Fanuc TP program (LS listing): hosenrohr_oVersatz.ls

/PROG  hosenrohr_oVersatz
/ATTR
COMMENT	= "19-03-19 17:34:17";
PROG_SIZE	= 0;
DEFAULT_GROUP	= 1, *, *, *, *;
/APPL
    ARC Welding Equipment: 1, *, *, *, *;
/MN
   1:  CALL HOME_ALL;
   1:  UFRAME_NUM = 1;
   1:  UTOOL_NUM = 3;
   1:  COL GUARD ADJUST 150;
   1:  PR[91] = PR[90];
   1:  PR[91,1] = PR[90,1] + 0.213;
   1:  PR[91,2] = PR[90,2] + 0.028;
   1:  PR[91,3] = PR[90,3] + 1.330;
   1:  PR[92] = PR[91];
   1:  PR[92,3] = PR[92,3] + 50;
   1:J PR[92] 10% FINE;
   1:L PR[91] R[100]mm/sec CNT100;
   1:  CALL LASER_DRAHT_START;
   1:  PR[91,1] = PR[90,1] + 0.684;
   1:  PR[91,2] = PR[90,2] + -0.011;
   1:L PR[91] R[100]mm/sec CNT100;
   1:  PR[91,1] = PR[90,1] + 1.247;
   1:  PR[91,2] = PR[90,2] + -0.156;
   1:  PR[91,3] = PR[90,3] + 0.003;
   1:L PR[91] R[100]mm/sec CNT100;
   1:  PR[91,1] = PR[90,1] + 1.774;
   1:  PR[91,2] = PR[90,2] + -0.407;
   1:  PR[91,3] = PR[90,3] + 0.006;
   1:L PR[91] R[100]mm/sec CNT100;
   1:  PR[91,1] = PR[90,1] + 2.182;
   1:  PR[91,2] = PR[90,2] + -0.695;
   1:  PR[91,3] = PR[90,3] + 0.010;
   1:L PR[91] R[100]mm/sec CNT100;
   1:  PR[91,1] = PR[90,1] + 2.537;
   1:  PR[91,2] = PR[90,2] + -1.047;
   1:  PR[91,3] = PR[90,3] + 0.013;
   1:L PR[91] R[100]mm/sec CNT100;
   1:  PR[91,1] = PR[90,1] + 2.876;
   1:  PR[91,2] = PR[90,2] + -1.521;
   1:  PR[91,3] = PR[90,3] + 0.016;
   1:L PR[91] R[100]mm/sec CNT100;
   1:  PR[91,1] = PR[90,1] + 3.117;
   1:  PR[91,2] = PR[90,2] + -2.049;
   1:  PR[91,3] = PR[90,3] + 0.020;
   1:L PR[91] R[100]mm/sec CNT100;
   1:  PR[91,1] = PR[90,1] + 3.228;
   1:  PR[91,2] = PR[90,2] + -2.464;
   1:  PR[91,3] = PR[90,3] + 0.023;
   1:L PR[91] R[100]mm/sec CNT100;
   1:  PR[91,1] = PR[90,1] + 3.332;
   1:  PR[91,2] = PR[90,2] + -2.996;
   1:  PR[91,3] = PR[90,3] + 0.026;
   1:L PR[91] R[100]mm/sec CNT100;
   1:  PR[91,1] = PR[90,1] + 3.499;
   1:  PR[91,2] = PR[90,2] + -3.723;
   1:  PR[91,3] = PR[90,3] + 0.029;
   1:L PR[91] R[100]mm/sec CNT100;
   1:  PR[91,1] = PR[90,1] + 3.811;
   1:  PR[91,2] = PR[90,2] + -4.797;
   1:  PR[91,3] = PR[90,3] + 0.034;
   1:L PR[91] R[100]mm/sec CNT100;
   1:  PR[91,1] = PR[90,1] + 4.268;
   1:  PR[91,2] = PR[90,2] + -6.041;
   1:  PR[91,3] = PR[90,3] + 0.040;
   1:L PR[91] R[100]mm/sec CNT100;
   1:  PR[91,1] = PR[90,1] + 4.777;
   1:  PR[91,2] = PR[90,2] + -7.153;
   1:  PR[91,3] = PR[90,3] + 0.048;
   1:L PR[91] R[100]mm/sec CNT100;
   1:  PR[91,1] = PR[90,1] + 5.314;
   1:  PR[91,2] = PR[90,2] + -8.138;
   1:  PR[91,3] = PR[90,3] + 0.056;
   1:L PR[91] R[100]mm/sec CNT100;
   1:  PR[91,1] = PR[90,1] + 5.705;
   1:  PR[91,2] = PR[90,2] + -8.772;
   1:  PR[91,3] = PR[90,3] + 0.063;
   1:L PR[91] R[100]mm/sec CNT100;
   1:  PR[91,1] = PR[90,1] + 6.024;
   1:  PR[91,2] = PR[90,2] + -9.246;
   1:  PR[91,3] = PR[90,3] + 0.067;
   1:L PR[91] R[100]mm/sec CNT100;
   1:  PR[91,1] = PR[90,1] + 6.762;
   1:  PR[91,2] = PR[90,2] + -10.226;
   1:  PR[91,3] = PR[90,3] + 0.071;
   1:L PR[91] R[100]mm/sec CNT100;
   1:  PR[91,1] = PR[90,1] + 7.570;
   1:  PR[91,2] = PR[90,2] + -11.150;
   1:  PR[91,3] = PR[90,3] + 0.078;
   1:L PR[91] R[100]mm/sec CNT100;
   1:  PR[91,1] = PR[90,1] + 8.074;
   1:  PR[91,2] = PR[90,2] + -11.664;
   1:  PR[91,3] = PR[90,3] + 0.086;
   1:L PR[91] R[100]mm/sec CNT100;
   1:  PR[91,1] = PR[90,1] + 8.430;
   1:  PR[91,2] = PR[90,2] + -12.001;
   1:  PR[91,3] = PR[90,3] + 0.090;
   1:L PR[91] R[100]mm/sec CNT100;
   1:  PR[91,1] = PR[90,1] + 9.365;
   1:  PR[91,2] = PR[90,2] + -12.801;
   1:  PR[91,3] = PR[90,3] + 0.093;
   1:L PR[91] R[100]mm/sec CNT100;
   1:  PR[91,1] = PR[90,1] + 10.262;
   1:  PR[91,2] = PR[90,2] + -13.466;
   1:  PR[91,3] = PR[90,3] + 0.100;
   1:L PR[91] R[100]mm/sec CNT100;
   1:  PR[91,1] = PR[90,1] + 11.385;
   1:  PR[91,2] = PR[90,2] + -14.181;
   1:  PR[91,3] = PR[90,3] + 0.107;
   1:L PR[91] R[100]mm/sec CNT100;
   1:  PR[91,1] = PR[90,1] + 12.079;
   1:  PR[91,2] = PR[90,2] + -14.564;
   1:  PR[91,3] = PR[90,3] + 0.115;
   1:L PR[91] R[100]mm/sec CNT100;
   1:  PR[91,1] = PR[90,1] + 12.452;
   1:  PR[91,2] = PR[90,2] + -14.752;
   1:  PR[91,3] = PR[90,3] + 0.120;
   1:L PR[91] R[100]mm/sec CNT100;
   1:  PR[91,1] = PR[90,1] + 13.575;
   1:  PR[91,2] = PR[90,2] + -15.252;
   1:  PR[91,3] = PR[90,3] + 0.123;
   1:L PR[91] R[100]mm/sec CNT100;
   1:  PR[91,1] = PR[90,1] + 14.627;
   1:  PR[91,2] = PR[90,2] + -15.633;
   1:  PR[91,3] = PR[90,3] + 0.130;
   1:L PR[91] R[100]mm/sec CNT100;
   1:  PR[91,1] = PR[90,1] + 15.902;
   1:  PR[91,2] = PR[90,2] + -15.997;
   1:  PR[91,3] = PR[90,3] + 0.137;
   1:L PR[91] R[100]mm/sec CNT100;
   1:  PR[91,1] = PR[90,1] + 17.100;
   1:  PR[91,2] = PR[90,2] + -16.242;
   1:  PR[91,3] = PR[90,3] + 0.145;
   1:L PR[91] R[100]mm/sec CNT100;
   1:  PR[91,1] = PR[90,1] + 18.207;
   1:  PR[91,2] = PR[90,2] + -16.387;
   1:  PR[91,3] = PR[90,3] + 0.152;
   1:L PR[91] R[100]mm/sec CNT100;
   1:  PR[91,1] = PR[90,1] + 19.533;
   1:  PR[91,2] = PR[90,2] + -16.468;
   1:  PR[91,3] = PR[90,3] + 0.159;
   1:L PR[91] R[100]mm/sec CNT100;
   1:  PR[91,1] = PR[90,1] + 20.752;
   1:  PR[91,2] = PR[90,2] + -16.449;
   1:  PR[91,3] = PR[90,3] + 0.167;
   1:L PR[91] R[100]mm/sec CNT100;
   1:  PR[91,1] = PR[90,1] + 21.868;
   1:  PR[91,2] = PR[90,2] + -16.353;
   1:  PR[91,3] = PR[90,3] + 0.175;
   1:L PR[91] R[100]mm/sec CNT100;
   1:  PR[91,1] = PR[90,1] + 23.177;
   1:  PR[91,2] = PR[90,2] + -16.147;
   1:  PR[91,3] = PR[90,3] + 0.181;
   1:L PR[91] R[100]mm/sec CNT100;
   1:  PR[91,1] = PR[90,1] + 24.367;
   1:  PR[91,2] = PR[90,2] + -15.866;
   1:  PR[91,3] = PR[90,3] + 0.189;
   1:L PR[91] R[100]mm/sec CNT100;
   1:  PR[91,1] = PR[90,1] + 25.433;
   1:  PR[91,2] = PR[90,2] + -15.532;
   1:  PR[91,3] = PR[90,3] + 0.197;
   1:L PR[91] R[100]mm/sec CNT100;
   1:  PR[91,1] = PR[90,1] + 26.669;
   1:  PR[91,2] = PR[90,2] + -15.048;
   1:  PR[91,3] = PR[90,3] + 0.204;
   1:L PR[91] R[100]mm/sec CNT100;
   1:  PR[91,1] = PR[90,1] + 27.769;
   1:  PR[91,2] = PR[90,2] + -14.518;
   1:  PR[91,3] = PR[90,3] + 0.212;
   1:L PR[91] R[100]mm/sec CNT100;
   1:  PR[91,1] = PR[90,1] + 28.829;
   1:  PR[91,2] = PR[90,2] + -13.909;
   1:  PR[91,3] = PR[90,3] + 0.219;
   1:L PR[91] R[100]mm/sec CNT100;
   1:  PR[91,1] = PR[90,1] + 29.757;
   1:  PR[91,2] = PR[90,2] + -13.284;
   1:  PR[91,3] = PR[90,3] + 0.227;
   1:L PR[91] R[100]mm/sec CNT100;
   1:  PR[91,1] = PR[90,1] + 30.802;
   1:  PR[91,2] = PR[90,2] + -12.468;
   1:  PR[91,3] = PR[90,3] + 0.233;
   1:L PR[91] R[100]mm/sec CNT100;
   1:  PR[91,1] = PR[90,1] + 31.706;
   1:  PR[91,2] = PR[90,2] + -11.646;
   1:  PR[91,3] = PR[90,3] + 0.241;
   1:L PR[91] R[100]mm/sec CNT100;
   1:  PR[91,1] = PR[90,1] + 32.547;
   1:  PR[91,2] = PR[90,2] + -10.760;
   1:  PR[91,3] = PR[90,3] + 0.249;
   1:L PR[91] R[100]mm/sec CNT100;
   1:  PR[91,1] = PR[90,1] + 33.259;
   1:  PR[91,2] = PR[90,2] + -9.896;
   1:  PR[91,3] = PR[90,3] + 0.256;
   1:L PR[91] R[100]mm/sec CNT100;
   1:  PR[91,1] = PR[90,1] + 34.054;
   1:  PR[91,2] = PR[90,2] + -8.776;
   1:  PR[91,3] = PR[90,3] + 0.263;
   1:L PR[91] R[100]mm/sec CNT100;
   1:  PR[91,1] = PR[90,1] + 34.659;
   1:  PR[91,2] = PR[90,2] + -7.769;
   1:  PR[91,3] = PR[90,3] + 0.271;
   1:L PR[91] R[100]mm/sec CNT100;
   1:  PR[91,1] = PR[90,1] + 35.214;
   1:  PR[91,2] = PR[90,2] + -6.678;
   1:  PR[91,3] = PR[90,3] + 0.279;
   1:L PR[91] R[100]mm/sec CNT100;
   1:  PR[91,1] = PR[90,1] + 35.547;
   1:  PR[91,2] = PR[90,2] + -5.910;
   1:  PR[91,3] = PR[90,3] + 0.286;
   1:L PR[91] R[100]mm/sec CNT100;
   1:  PR[91,1] = PR[90,1] + 35.684;
   1:  PR[91,2] = PR[90,2] + -5.559;
   1:  PR[91,3] = PR[90,3] + 0.291;
   1:L PR[91] R[100]mm/sec CNT100;
   1:  PR[91,1] = PR[90,1] + 36.077;
   1:  PR[91,2] = PR[90,2] + -4.396;
   1:  PR[91,3] = PR[90,3] + 0.293;
   1:L PR[91] R[100]mm/sec CNT100;
   1:  PR[91,1] = PR[90,1] + 36.362;
   1:  PR[91,2] = PR[90,2] + -3.304;
   1:  PR[91,3] = PR[90,3] + 0.301;
   1:L PR[91] R[100]mm/sec CNT100;
   1:  PR[91,1] = PR[90,1] + 36.446;
   1:  PR[91,2] = PR[90,2] + -2.914;
   1:  PR[91,3] = PR[90,3] + 0.308;
   1:L PR[91] R[100]mm/sec CNT100;
   1:  PR[91,1] = PR[90,1] + 36.603;
   1:  PR[91,2] = PR[90,2] + -2.012;
   1:  PR[91,3] = PR[90,3] + 0.310;
   1:L PR[91] R[100]mm/sec CNT100;
   1:  PR[91,1] = PR[90,1] + 36.727;
   1:  PR[91,2] = PR[90,2] + -0.896;
   1:  PR[91,3] = PR[90,3] + 0.316;
   1:L PR[91] R[100]mm/sec CNT100;
   1:  PR[91,1] = PR[90,1] + 36.773;
   1:  PR[91,2] = PR[90,2] + -0.086;
   1:  PR[91,3] = PR[90,3] + 0.322;
   1:L PR[91] R[100]mm/sec CNT100;
   1:  PR[91,1] = PR[90,1] + 36.781;
   1:  PR[91,2] = PR[90,2] + 0.420;
   1:  PR[91,3] = PR[90,3] + 0.327;
   1:L PR[91] R[100]mm/sec CNT100;
   1:  PR[91,1] = PR[90,1] + 36.726;
   1:  PR[91,2] = PR[90,2] + 1.756;
   1:  PR[91,3] = PR[90,3] + 0.330;
   1:L PR[91] R[100]mm/sec CNT100;
   1:  PR[91,1] = PR[90,1] + 36.604;
   1:  PR[91,2] = PR[90,2] + 2.865;
   1:  PR[91,3] = PR[90,3] + 0.339;
   1:L PR[91] R[100]mm/sec CNT100;
   1:  PR[91,1] = PR[90,1] + 36.404;
   1:  PR[91,2] = PR[90,2] + 3.965;
   1:  PR[91,3] = PR[90,3] + 0.345;
   1:L PR[91] R[100]mm/sec CNT100;
   1:  PR[91,1] = PR[90,1] + 36.075;
   1:  PR[91,2] = PR[90,2] + 5.258;
   1:  PR[91,3] = PR[90,3] + 0.352;
   1:L PR[91] R[100]mm/sec CNT100;
   1:  PR[91,1] = PR[90,1] + 35.922;
   1:  PR[91,2] = PR[90,2] + 5.747;
   1:  PR[91,3] = PR[90,3] + 0.360;
   1:L PR[91] R[100]mm/sec CNT100;
   1:  PR[91,1] = PR[90,1] + 35.650;
   1:  PR[91,2] = PR[90,2] + 6.499;
   1:  PR[91,3] = PR[90,3] + 0.363;
   1:L PR[91] R[100]mm/sec CNT100;
   1:  PR[91,1] = PR[90,1] + 35.212;
   1:  PR[91,2] = PR[90,2] + 7.536;
   1:  PR[91,3] = PR[90,3] + 0.368;
   1:L PR[91] R[100]mm/sec CNT100;
   1:  PR[91,1] = PR[90,1] + 34.705;
   1:  PR[91,2] = PR[90,2] + 8.538;
   1:  PR[91,3] = PR[90,3] + 0.375;
   1:L PR[91] R[100]mm/sec CNT100;
   1:  PR[91,1] = PR[90,1] + 34.027;
   1:  PR[91,2] = PR[90,2] + 9.673;
   1:  PR[91,3] = PR[90,3] + 0.382;
   1:L PR[91] R[100]mm/sec CNT100;
   1:  PR[91,1] = PR[90,1] + 33.322;
   1:  PR[91,2] = PR[90,2] + 10.671;
   1:  PR[91,3] = PR[90,3] + 0.390;
   1:L PR[91] R[100]mm/sec CNT100;
   1:  PR[91,1] = PR[90,1] + 32.675;
   1:  PR[91,2] = PR[90,2] + 11.466;
   1:  PR[91,3] = PR[90,3] + 0.397;
   1:L PR[91] R[100]mm/sec CNT100;
   1:  PR[91,1] = PR[90,1] + 31.777;
   1:  PR[91,2] = PR[90,2] + 12.428;
   1:  PR[91,3] = PR[90,3] + 0.404;
   1:L PR[91] R[100]mm/sec CNT100;
   1:  PR[91,1] = PR[90,1] + 30.801;
   1:  PR[91,2] = PR[90,2] + 13.325;
   1:  PR[91,3] = PR[90,3] + 0.412;
   1:L PR[91] R[100]mm/sec CNT100;
   1:  PR[91,1] = PR[90,1] + 29.837;
   1:  PR[91,2] = PR[90,2] + 14.083;
   1:  PR[91,3] = PR[90,3] + 0.420;
   1:L PR[91] R[100]mm/sec CNT100;
   1:  PR[91,1] = PR[90,1] + 29.332;
   1:  PR[91,2] = PR[90,2] + 14.438;
   1:  PR[91,3] = PR[90,3] + 0.427;
   1:L PR[91] R[100]mm/sec CNT100;
   1:  PR[91,1] = PR[90,1] + 28.834;
   1:  PR[91,2] = PR[90,2] + 14.760;
   1:  PR[91,3] = PR[90,3] + 0.431;
   1:L PR[91] R[100]mm/sec CNT100;
   1:  PR[91,1] = PR[90,1] + 27.676;
   1:  PR[91,2] = PR[90,2] + 15.420;
   1:  PR[91,3] = PR[90,3] + 0.434;
   1:L PR[91] R[100]mm/sec CNT100;
   1:  PR[91,1] = PR[90,1] + 26.668;
   1:  PR[91,2] = PR[90,2] + 15.904;
   1:  PR[91,3] = PR[90,3] + 0.442;
   1:L PR[91] R[100]mm/sec CNT100;
   1:  PR[91,1] = PR[90,1] + 25.628;
   1:  PR[91,2] = PR[90,2] + 16.318;
   1:  PR[91,3] = PR[90,3] + 0.449;
   1:L PR[91] R[100]mm/sec CNT100;
   1:  PR[91,1] = PR[90,1] + 24.365;
   1:  PR[91,2] = PR[90,2] + 16.721;
   1:  PR[91,3] = PR[90,3] + 0.456;
   1:L PR[91] R[100]mm/sec CNT100;
   1:  PR[91,1] = PR[90,1] + 23.177;
   1:  PR[91,2] = PR[90,2] + 17.002;
   1:  PR[91,3] = PR[90,3] + 0.464;
   1:L PR[91] R[100]mm/sec CNT100;
   1:  PR[91,1] = PR[90,1] + 21.868;
   1:  PR[91,2] = PR[90,2] + 17.208;
   1:  PR[91,3] = PR[90,3] + 0.472;
   1:L PR[91] R[100]mm/sec CNT100;
   1:  PR[91,1] = PR[90,1] + 20.752;
   1:  PR[91,2] = PR[90,2] + 17.305;
   1:  PR[91,3] = PR[90,3] + 0.480;
   1:L PR[91] R[100]mm/sec CNT100;
   1:  PR[91,1] = PR[90,1] + 19.634;
   1:  PR[91,2] = PR[90,2] + 17.324;
   1:  PR[91,3] = PR[90,3] + 0.486;
   1:L PR[91] R[100]mm/sec CNT100;
   1:  PR[91,1] = PR[90,1] + 18.412;
   1:  PR[91,2] = PR[90,2] + 17.261;
   1:  PR[91,3] = PR[90,3] + 0.493;
   1:L PR[91] R[100]mm/sec CNT100;
   1:  PR[91,1] = PR[90,1] + 17.098;
   1:  PR[91,2] = PR[90,2] + 17.096;
   1:  PR[91,3] = PR[90,3] + 0.501;
   1:L PR[91] R[100]mm/sec CNT100;
   1:  PR[91,1] = PR[90,1] + 15.901;
   1:  PR[91,2] = PR[90,2] + 16.852;
   1:  PR[91,3] = PR[90,3] + 0.509;
   1:L PR[91] R[100]mm/sec CNT100;
   1:  PR[91,1] = PR[90,1] + 14.725;
   1:  PR[91,2] = PR[90,2] + 16.521;
   1:  PR[91,3] = PR[90,3] + 0.516;
   1:L PR[91] R[100]mm/sec CNT100;
   1:  PR[91,1] = PR[90,1] + 13.575;
   1:  PR[91,2] = PR[90,2] + 16.106;
   1:  PR[91,3] = PR[90,3] + 0.524;
   1:L PR[91] R[100]mm/sec CNT100;
   1:  PR[91,1] = PR[90,1] + 12.458;
   1:  PR[91,2] = PR[90,2] + 15.610;
   1:  PR[91,3] = PR[90,3] + 0.531;
   1:L PR[91] R[100]mm/sec CNT100;
   1:  PR[91,1] = PR[90,1] + 11.381;
   1:  PR[91,2] = PR[90,2] + 15.034;
   1:  PR[91,3] = PR[90,3] + 0.538;
   1:L PR[91] R[100]mm/sec CNT100;
   1:  PR[91,1] = PR[90,1] + 10.348;
   1:  PR[91,2] = PR[90,2] + 14.382;
   1:  PR[91,3] = PR[90,3] + 0.546;
   1:L PR[91] R[100]mm/sec CNT100;
   1:  PR[91,1] = PR[90,1] + 9.286;
   1:  PR[91,2] = PR[90,2] + 13.591;
   1:  PR[91,3] = PR[90,3] + 0.553;
   1:L PR[91] R[100]mm/sec CNT100;
   1:  PR[91,1] = PR[90,1] + 8.360;
   1:  PR[91,2] = PR[90,2] + 12.790;
   1:  PR[91,3] = PR[90,3] + 0.561;
   1:L PR[91] R[100]mm/sec CNT100;
   1:  PR[91,1] = PR[90,1] + 7.564;
   1:  PR[91,2] = PR[90,2] + 11.999;
   1:  PR[91,3] = PR[90,3] + 0.569;
   1:L PR[91] R[100]mm/sec CNT100;
   1:  PR[91,1] = PR[90,1] + 7.149;
   1:  PR[91,2] = PR[90,2] + 11.541;
   1:  PR[91,3] = PR[90,3] + 0.576;
   1:L PR[91] R[100]mm/sec CNT100;
   1:  PR[91,1] = PR[90,1] + 6.702;
   1:  PR[91,2] = PR[90,2] + 11.004;
   1:  PR[91,3] = PR[90,3] + 0.579;
   1:L PR[91] R[100]mm/sec CNT100;
   1:  PR[91,1] = PR[90,1] + 6.028;
   1:  PR[91,2] = PR[90,2] + 10.107;
   1:  PR[91,3] = PR[90,3] + 0.584;
   1:L PR[91] R[100]mm/sec CNT100;
   1:  PR[91,1] = PR[90,1] + 5.360;
   1:  PR[91,2] = PR[90,2] + 9.073;
   1:  PR[91,3] = PR[90,3] + 0.590;
   1:L PR[91] R[100]mm/sec CNT100;
   1:  PR[91,1] = PR[90,1] + 5.101;
   1:  PR[91,2] = PR[90,2] + 8.622;
   1:  PR[91,3] = PR[90,3] + 0.598;
   1:L PR[91] R[100]mm/sec CNT100;
   1:  PR[91,1] = PR[90,1] + 4.779;
   1:  PR[91,2] = PR[90,2] + 8.013;
   1:  PR[91,3] = PR[90,3] + 0.601;
   1:L PR[91] R[100]mm/sec CNT100;
   1:  PR[91,1] = PR[90,1] + 4.230;
   1:  PR[91,2] = PR[90,2] + 6.799;
   1:  PR[91,3] = PR[90,3] + 0.605;
   1:L PR[91] R[100]mm/sec CNT100;
   1:  PR[91,1] = PR[90,1] + 3.836;
   1:  PR[91,2] = PR[90,2] + 5.734;
   1:  PR[91,3] = PR[90,3] + 0.613;
   1:L PR[91] R[100]mm/sec CNT100;
   1:  PR[91,1] = PR[90,1] + 3.527;
   1:  PR[91,2] = PR[90,2] + 4.682;
   1:  PR[91,3] = PR[90,3] + 0.620;
   1:L PR[91] R[100]mm/sec CNT100;
   1:  PR[91,1] = PR[90,1] + 3.234;
   1:  PR[91,2] = PR[90,2] + 3.348;
   1:  PR[91,3] = PR[90,3] + 0.627;
   1:L PR[91] R[100]mm/sec CNT100;
   1:  PR[91,1] = PR[90,1] + 3.105;
   1:  PR[91,2] = PR[90,2] + 2.866;
   1:  PR[91,3] = PR[90,3] + 0.635;
   1:L PR[91] R[100]mm/sec CNT100;
   1:  PR[91,1] = PR[90,1] + 2.875;
   1:  PR[91,2] = PR[90,2] + 2.376;
   1:  PR[91,3] = PR[90,3] + 0.638;
   1:L PR[91] R[100]mm/sec CNT100;
   1:  PR[91,1] = PR[90,1] + 2.564;
   1:  PR[91,2] = PR[90,2] + 1.931;
   1:  PR[91,3] = PR[90,3] + 0.641;
   1:L PR[91] R[100]mm/sec CNT100;
   1:  PR[91,1] = PR[90,1] + 2.183;
   1:  PR[91,2] = PR[90,2] + 1.551;
   1:  PR[91,3] = PR[90,3] + 0.645;
   1:L PR[91] R[100]mm/sec CNT100;
   1:  PR[91,1] = PR[90,1] + 1.771;
   1:  PR[91,2] = PR[90,2] + 1.260;
   1:  PR[91,3] = PR[90,3] + 0.648;
   1:L PR[91] R[100]mm/sec CNT100;
   1:  PR[91,1] = PR[90,1] + 1.212;
   1:  PR[91,2] = PR[90,2] + 1.000;
   1:  PR[91,3] = PR[90,3] + 0.651;
   1:L PR[91] R[100]mm/sec CNT100;
   1:  PR[91,1] = PR[90,1] + 0.724;
   1:  PR[91,2] = PR[90,2] + 0.872;
   1:  PR[91,3] = PR[90,3] + 0.655;
   1:L PR[91] R[100]mm/sec CNT100;
   1:  PR[91,1] = PR[90,1] + 0.253;
   1:  PR[91,2] = PR[90,2] + 0.829;
   1:  PR[91,3] = PR[90,3] + 0.658;
   1:L PR[91] R[100]mm/sec CNT100;
   1:  PR[91,1] = PR[90,1] + -0.453;
   1:  PR[91,2] = PR[90,2] + 0.828;
   1:  PR[91,3] = PR[90,3] + 0.661;
   1:L PR[91] R[100]mm/sec CNT100;
   1:  PR[91,1] = PR[90,1] + -0.963;
   1:  PR[91,2] = PR[90,2] + 0.871;
   1:  PR[91,3] = PR[90,3] + 0.665;
   1:L PR[91] R[100]mm/sec CNT100;
   1:  PR[91,1] = PR[90,1] + -1.489;
   1:  PR[91,2] = PR[90,2] + 1.013;
   1:  PR[91,3] = PR[90,3] + 0.668;
   1:L PR[91] R[100]mm/sec CNT100;
   1:  PR[91,1] = PR[90,1] + -2.012;
   1:  PR[91,2] = PR[90,2] + 1.262;
   1:  PR[91,3] = PR[90,3] + 0.671;
   1:L PR[91] R[100]mm/sec CNT100;
   1:  PR[91,1] = PR[90,1] + -2.421;
   1:  PR[91,2] = PR[90,2] + 1.550;
   1:  PR[91,3] = PR[90,3] + 0.675;
   1:L PR[91] R[100]mm/sec CNT100;
   1:  PR[91,1] = PR[90,1] + -2.775;
   1:  PR[91,2] = PR[90,2] + 1.902;
   1:  PR[91,3] = PR[90,3] + 0.678;
   1:L PR[91] R[100]mm/sec CNT100;
   1:  PR[91,1] = PR[90,1] + -3.106;
   1:  PR[91,2] = PR[90,2] + 2.365;
   1:  PR[91,3] = PR[90,3] + 0.681;
   1:L PR[91] R[100]mm/sec CNT100;
   1:  PR[91,1] = PR[90,1] + -3.257;
   1:  PR[91,2] = PR[90,2] + 2.660;
   1:  PR[91,3] = PR[90,3] + 0.684;
   1:L PR[91] R[100]mm/sec CNT100;
   1:  PR[91,1] = PR[90,1] + -3.359;
   1:  PR[91,2] = PR[90,2] + 2.920;
   1:  PR[91,3] = PR[90,3] + 0.686;
   1:L PR[91] R[100]mm/sec CNT100;
   1:  PR[91,1] = PR[90,1] + -3.465;
   1:  PR[91,2] = PR[90,2] + 3.314;
   1:  PR[91,3] = PR[90,3] + 0.688;
   1:L PR[91] R[100]mm/sec CNT100;
   1:  PR[91,1] = PR[90,1] + -3.738;
   1:  PR[91,2] = PR[90,2] + 4.582;
   1:  PR[91,3] = PR[90,3] + 0.691;
   1:L PR[91] R[100]mm/sec CNT100;
   1:  PR[91,1] = PR[90,1] + -4.049;
   1:  PR[91,2] = PR[90,2] + 5.652;
   1:  PR[91,3] = PR[90,3] + 0.699;
   1:L PR[91] R[100]mm/sec CNT100;
   1:  PR[91,1] = PR[90,1] + -4.507;
   1:  PR[91,2] = PR[90,2] + 6.896;
   1:  PR[91,3] = PR[90,3] + 0.705;
   1:L PR[91] R[100]mm/sec CNT100;
   1:  PR[91,1] = PR[90,1] + -5.017;
   1:  PR[91,2] = PR[90,2] + 8.012;
   1:  PR[91,3] = PR[90,3] + 0.713;
   1:L PR[91] R[100]mm/sec CNT100;
   1:  PR[91,1] = PR[90,1] + -5.339;
   1:  PR[91,2] = PR[90,2] + 8.622;
   1:  PR[91,3] = PR[90,3] + 0.721;
   1:L PR[91] R[100]mm/sec CNT100;
   1:  PR[91,1] = PR[90,1] + -5.598;
   1:  PR[91,2] = PR[90,2] + 9.073;
   1:  PR[91,3] = PR[90,3] + 0.725;
   1:L PR[91] R[100]mm/sec CNT100;
   1:  PR[91,1] = PR[90,1] + -6.266;
   1:  PR[91,2] = PR[90,2] + 10.106;
   1:  PR[91,3] = PR[90,3] + 0.728;
   1:L PR[91] R[100]mm/sec CNT100;
   1:  PR[91,1] = PR[90,1] + -7.004;
   1:  PR[91,2] = PR[90,2] + 11.085;
   1:  PR[91,3] = PR[90,3] + 0.736;
   1:L PR[91] R[100]mm/sec CNT100;
   1:  PR[91,1] = PR[90,1] + -7.387;
   1:  PR[91,2] = PR[90,2] + 11.540;
   1:  PR[91,3] = PR[90,3] + 0.743;
   1:L PR[91] R[100]mm/sec CNT100;
   1:  PR[91,1] = PR[90,1] + -7.802;
   1:  PR[91,2] = PR[90,2] + 11.998;
   1:  PR[91,3] = PR[90,3] + 0.747;
   1:L PR[91] R[100]mm/sec CNT100;
   1:  PR[91,1] = PR[90,1] + -8.673;
   1:  PR[91,2] = PR[90,2] + 12.861;
   1:  PR[91,3] = PR[90,3] + 0.750;
   1:L PR[91] R[100]mm/sec CNT100;
   1:  PR[91,1] = PR[90,1] + -9.603;
   1:  PR[91,2] = PR[90,2] + 13.656;
   1:  PR[91,3] = PR[90,3] + 0.758;
   1:L PR[91] R[100]mm/sec CNT100;
   1:  PR[91,1] = PR[90,1] + -10.501;
   1:  PR[91,2] = PR[90,2] + 14.321;
   1:  PR[91,3] = PR[90,3] + 0.765;
   1:L PR[91] R[100]mm/sec CNT100;
   1:  PR[91,1] = PR[90,1] + -11.621;
   1:  PR[91,2] = PR[90,2] + 15.034;
   1:  PR[91,3] = PR[90,3] + 0.772;
   1:L PR[91] R[100]mm/sec CNT100;
   1:  PR[91,1] = PR[90,1] + -12.697;
   1:  PR[91,2] = PR[90,2] + 15.610;
   1:  PR[91,3] = PR[90,3] + 0.780;
   1:L PR[91] R[100]mm/sec CNT100;
   1:  PR[91,1] = PR[90,1] + -13.814;
   1:  PR[91,2] = PR[90,2] + 16.107;
   1:  PR[91,3] = PR[90,3] + 0.788;
   1:L PR[91] R[100]mm/sec CNT100;
   1:  PR[91,1] = PR[90,1] + -14.866;
   1:  PR[91,2] = PR[90,2] + 16.488;
   1:  PR[91,3] = PR[90,3] + 0.795;
   1:L PR[91] R[100]mm/sec CNT100;
   1:  PR[91,1] = PR[90,1] + -16.141;
   1:  PR[91,2] = PR[90,2] + 16.852;
   1:  PR[91,3] = PR[90,3] + 0.802;
   1:L PR[91] R[100]mm/sec CNT100;
   1:  PR[91,1] = PR[90,1] + -17.338;
   1:  PR[91,2] = PR[90,2] + 17.097;
   1:  PR[91,3] = PR[90,3] + 0.810;
   1:L PR[91] R[100]mm/sec CNT100;
   1:  PR[91,1] = PR[90,1] + -18.446;
   1:  PR[91,2] = PR[90,2] + 17.242;
   1:  PR[91,3] = PR[90,3] + 0.817;
   1:L PR[91] R[100]mm/sec CNT100;
   1:  PR[91,1] = PR[90,1] + -19.771;
   1:  PR[91,2] = PR[90,2] + 17.323;
   1:  PR[91,3] = PR[90,3] + 0.824;
   1:L PR[91] R[100]mm/sec CNT100;
   1:  PR[91,1] = PR[90,1] + -20.991;
   1:  PR[91,2] = PR[90,2] + 17.305;
   1:  PR[91,3] = PR[90,3] + 0.832;
   1:L PR[91] R[100]mm/sec CNT100;
   1:  PR[91,1] = PR[90,1] + -22.107;
   1:  PR[91,2] = PR[90,2] + 17.208;
   1:  PR[91,3] = PR[90,3] + 0.840;
   1:L PR[91] R[100]mm/sec CNT100;
   1:  PR[91,1] = PR[90,1] + -23.415;
   1:  PR[91,2] = PR[90,2] + 17.002;
   1:  PR[91,3] = PR[90,3] + 0.846;
   1:L PR[91] R[100]mm/sec CNT100;
   1:  PR[91,1] = PR[90,1] + -24.605;
   1:  PR[91,2] = PR[90,2] + 16.721;
   1:  PR[91,3] = PR[90,3] + 0.854;
   1:L PR[91] R[100]mm/sec CNT100;
   1:  PR[91,1] = PR[90,1] + -25.770;
   1:  PR[91,2] = PR[90,2] + 16.355;
   1:  PR[91,3] = PR[90,3] + 0.862;
   1:L PR[91] R[100]mm/sec CNT100;
   1:  PR[91,1] = PR[90,1] + -26.907;
   1:  PR[91,2] = PR[90,2] + 15.904;
   1:  PR[91,3] = PR[90,3] + 0.869;
   1:L PR[91] R[100]mm/sec CNT100;
   1:  PR[91,1] = PR[90,1] + -27.915;
   1:  PR[91,2] = PR[90,2] + 15.420;
   1:  PR[91,3] = PR[90,3] + 0.877;
   1:L PR[91] R[100]mm/sec CNT100;
   1:  PR[91,1] = PR[90,1] + -28.984;
   1:  PR[91,2] = PR[90,2] + 14.813;
   1:  PR[91,3] = PR[90,3] + 0.883;
   1:L PR[91] R[100]mm/sec CNT100;
   1:  PR[91,1] = PR[90,1] + -29.571;
   1:  PR[91,2] = PR[90,2] + 14.437;
   1:  PR[91,3] = PR[90,3] + 0.891;
   1:L PR[91] R[100]mm/sec CNT100;
   1:  PR[91,1] = PR[90,1] + -30.076;
   1:  PR[91,2] = PR[90,2] + 14.083;
   1:  PR[91,3] = PR[90,3] + 0.895;
   1:L PR[91] R[100]mm/sec CNT100;
   1:  PR[91,1] = PR[90,1] + -31.040;
   1:  PR[91,2] = PR[90,2] + 13.324;
   1:  PR[91,3] = PR[90,3] + 0.899;
   1:L PR[91] R[100]mm/sec CNT100;
   1:  PR[91,1] = PR[90,1] + -31.945;
   1:  PR[91,2] = PR[90,2] + 12.500;
   1:  PR[91,3] = PR[90,3] + 0.906;
   1:L PR[91] R[100]mm/sec CNT100;
   1:  PR[91,1] = PR[90,1] + -32.715;
   1:  PR[91,2] = PR[90,2] + 11.692;
   1:  PR[91,3] = PR[90,3] + 0.914;
   1:L PR[91] R[100]mm/sec CNT100;
   1:  PR[91,1] = PR[90,1] + -33.562;
   1:  PR[91,2] = PR[90,2] + 10.668;
   1:  PR[91,3] = PR[90,3] + 0.921;
   1:L PR[91] R[100]mm/sec CNT100;
   1:  PR[91,1] = PR[90,1] + -34.266;
   1:  PR[91,2] = PR[90,2] + 9.672;
   1:  PR[91,3] = PR[90,3] + 0.929;
   1:L PR[91] R[100]mm/sec CNT100;
   1:  PR[91,1] = PR[90,1] + -34.895;
   1:  PR[91,2] = PR[90,2] + 8.629;
   1:  PR[91,3] = PR[90,3] + 0.936;
   1:L PR[91] R[100]mm/sec CNT100;
   1:  PR[91,1] = PR[90,1] + -35.451;
   1:  PR[91,2] = PR[90,2] + 7.536;
   1:  PR[91,3] = PR[90,3] + 0.943;
   1:L PR[91] R[100]mm/sec CNT100;
   1:  PR[91,1] = PR[90,1] + -35.889;
   1:  PR[91,2] = PR[90,2] + 6.499;
   1:  PR[91,3] = PR[90,3] + 0.951;
   1:L PR[91] R[100]mm/sec CNT100;
   1:  PR[91,1] = PR[90,1] + -36.160;
   1:  PR[91,2] = PR[90,2] + 5.747;
   1:  PR[91,3] = PR[90,3] + 0.958;
   1:L PR[91] R[100]mm/sec CNT100;
   1:  PR[91,1] = PR[90,1] + -36.314;
   1:  PR[91,2] = PR[90,2] + 5.257;
   1:  PR[91,3] = PR[90,3] + 0.963;
   1:L PR[91] R[100]mm/sec CNT100;
   1:  PR[91,1] = PR[90,1] + -36.598;
   1:  PR[91,2] = PR[90,2] + 4.169;
   1:  PR[91,3] = PR[90,3] + 0.966;
   1:L PR[91] R[100]mm/sec CNT100;
   1:  PR[91,1] = PR[90,1] + -36.860;
   1:  PR[91,2] = PR[90,2] + 2.732;
   1:  PR[91,3] = PR[90,3] + 0.973;
   1:L PR[91] R[100]mm/sec CNT100;
   1:  PR[91,1] = PR[90,1] + -36.974;
   1:  PR[91,2] = PR[90,2] + 1.653;
   1:  PR[91,3] = PR[90,3] + 0.981;
   1:L PR[91] R[100]mm/sec CNT100;
   1:  PR[91,1] = PR[90,1] + -37.019;
   1:  PR[91,2] = PR[90,2] + 0.421;
   1:  PR[91,3] = PR[90,3] + 0.988;
   1:L PR[91] R[100]mm/sec CNT100;
   1:  PR[91,1] = PR[90,1] + -37.011;
   1:  PR[91,2] = PR[90,2] + -0.088;
   1:  PR[91,3] = PR[90,3] + 0.996;
   1:L PR[91] R[100]mm/sec CNT100;
   1:  PR[91,1] = PR[90,1] + -36.975;
   1:  PR[91,2] = PR[90,2] + -0.793;
   1:  PR[91,3] = PR[90,3] + 0.999;
   1:L PR[91] R[100]mm/sec CNT100;
   1:  PR[91,1] = PR[90,1] + -36.855;
   1:  PR[91,2] = PR[90,2] + -1.910;
   1:  PR[91,3] = PR[90,3] + 1.003;
   1:L PR[91] R[100]mm/sec CNT100;
   1:  PR[91,1] = PR[90,1] + -36.684;
   1:  PR[91,2] = PR[90,2] + -2.916;
   1:  PR[91,3] = PR[90,3] + 1.010;
   1:L PR[91] R[100]mm/sec CNT100;
   1:  PR[91,1] = PR[90,1] + -36.600;
   1:  PR[91,2] = PR[90,2] + -3.304;
   1:  PR[91,3] = PR[90,3] + 1.016;
   1:L PR[91] R[100]mm/sec CNT100;
   1:  PR[91,1] = PR[90,1] + -36.316;
   1:  PR[91,2] = PR[90,2] + -4.396;
   1:  PR[91,3] = PR[90,3] + 1.018;
   1:L PR[91] R[100]mm/sec CNT100;
   1:  PR[91,1] = PR[90,1] + -35.925;
   1:  PR[91,2] = PR[90,2] + -5.553;
   1:  PR[91,3] = PR[90,3] + 1.025;
   1:L PR[91] R[100]mm/sec CNT100;
   1:  PR[91,1] = PR[90,1] + -35.451;
   1:  PR[91,2] = PR[90,2] + -6.681;
   1:  PR[91,3] = PR[90,3] + 1.033;
   1:L PR[91] R[100]mm/sec CNT100;
   1:  PR[91,1] = PR[90,1] + -34.947;
   1:  PR[91,2] = PR[90,2] + -7.676;
   1:  PR[91,3] = PR[90,3] + 1.040;
   1:L PR[91] R[100]mm/sec CNT100;
   1:  PR[91,1] = PR[90,1] + -34.207;
   1:  PR[91,2] = PR[90,2] + -8.904;
   1:  PR[91,3] = PR[90,3] + 1.047;
   1:L PR[91] R[100]mm/sec CNT100;
   1:  PR[91,1] = PR[90,1] + -33.623;
   1:  PR[91,2] = PR[90,2] + -9.730;
   1:  PR[91,3] = PR[90,3] + 1.056;
   1:L PR[91] R[100]mm/sec CNT100;
   1:  PR[91,1] = PR[90,1] + -32.785;
   1:  PR[91,2] = PR[90,2] + -10.761;
   1:  PR[91,3] = PR[90,3] + 1.062;
   1:L PR[91] R[100]mm/sec CNT100;
   1:  PR[91,1] = PR[90,1] + -31.923;
   1:  PR[91,2] = PR[90,2] + -11.666;
   1:  PR[91,3] = PR[90,3] + 1.070;
   1:L PR[91] R[100]mm/sec CNT100;
   1:  PR[91,1] = PR[90,1] + -31.040;
   1:  PR[91,2] = PR[90,2] + -12.469;
   1:  PR[91,3] = PR[90,3] + 1.077;
   1:L PR[91] R[100]mm/sec CNT100;
   1:  PR[91,1] = PR[90,1] + -30.080;
   1:  PR[91,2] = PR[90,2] + -13.225;
   1:  PR[91,3] = PR[90,3] + 1.085;
   1:L PR[91] R[100]mm/sec CNT100;
   1:  PR[91,1] = PR[90,1] + -29.067;
   1:  PR[91,2] = PR[90,2] + -13.909;
   1:  PR[91,3] = PR[90,3] + 1.092;
   1:L PR[91] R[100]mm/sec CNT100;
   1:  PR[91,1] = PR[90,1] + -28.007;
   1:  PR[91,2] = PR[90,2] + -14.518;
   1:  PR[91,3] = PR[90,3] + 1.099;
   1:L PR[91] R[100]mm/sec CNT100;
   1:  PR[91,1] = PR[90,1] + -26.907;
   1:  PR[91,2] = PR[90,2] + -15.049;
   1:  PR[91,3] = PR[90,3] + 1.107;
   1:L PR[91] R[100]mm/sec CNT100;
   1:  PR[91,1] = PR[90,1] + -25.770;
   1:  PR[91,2] = PR[90,2] + -15.499;
   1:  PR[91,3] = PR[90,3] + 1.114;
   1:L PR[91] R[100]mm/sec CNT100;
   1:  PR[91,1] = PR[90,1] + -24.605;
   1:  PR[91,2] = PR[90,2] + -15.866;
   1:  PR[91,3] = PR[90,3] + 1.122;
   1:L PR[91] R[100]mm/sec CNT100;
   1:  PR[91,1] = PR[90,1] + -23.414;
   1:  PR[91,2] = PR[90,2] + -16.148;
   1:  PR[91,3] = PR[90,3] + 1.129;
   1:L PR[91] R[100]mm/sec CNT100;
   1:  PR[91,1] = PR[90,1] + -22.209;
   1:  PR[91,2] = PR[90,2] + -16.342;
   1:  PR[91,3] = PR[90,3] + 1.137;
   1:L PR[91] R[100]mm/sec CNT100;
   1:  PR[91,1] = PR[90,1] + -20.990;
   1:  PR[91,2] = PR[90,2] + -16.449;
   1:  PR[91,3] = PR[90,3] + 1.144;
   1:L PR[91] R[100]mm/sec CNT100;
   1:  PR[91,1] = PR[90,1] + -19.770;
   1:  PR[91,2] = PR[90,2] + -16.468;
   1:  PR[91,3] = PR[90,3] + 1.151;
   1:L PR[91] R[100]mm/sec CNT100;
   1:  PR[91,1] = PR[90,1] + -18.548;
   1:  PR[91,2] = PR[90,2] + -16.399;
   1:  PR[91,3] = PR[90,3] + 1.159;
   1:L PR[91] R[100]mm/sec CNT100;
   1:  PR[91,1] = PR[90,1] + -17.339;
   1:  PR[91,2] = PR[90,2] + -16.242;
   1:  PR[91,3] = PR[90,3] + 1.166;
   1:L PR[91] R[100]mm/sec CNT100;
   1:  PR[91,1] = PR[90,1] + -16.039;
   1:  PR[91,2] = PR[90,2] + -15.970;
   1:  PR[91,3] = PR[90,3] + 1.174;
   1:L PR[91] R[100]mm/sec CNT100;
   1:  PR[91,1] = PR[90,1] + -14.964;
   1:  PR[91,2] = PR[90,2] + -15.667;
   1:  PR[91,3] = PR[90,3] + 1.182;
   1:L PR[91] R[100]mm/sec CNT100;
   1:  PR[91,1] = PR[90,1] + -13.814;
   1:  PR[91,2] = PR[90,2] + -15.251;
   1:  PR[91,3] = PR[90,3] + 1.189;
   1:L PR[91] R[100]mm/sec CNT100;
   1:  PR[91,1] = PR[90,1] + -12.690;
   1:  PR[91,2] = PR[90,2] + -14.752;
   1:  PR[91,3] = PR[90,3] + 1.196;
   1:L PR[91] R[100]mm/sec CNT100;
   1:  PR[91,1] = PR[90,1] + -12.317;
   1:  PR[91,2] = PR[90,2] + -14.563;
   1:  PR[91,3] = PR[90,3] + 1.203;
   1:L PR[91] R[100]mm/sec CNT100;
   1:  PR[91,1] = PR[90,1] + -11.623;
   1:  PR[91,2] = PR[90,2] + -14.181;
   1:  PR[91,3] = PR[90,3] + 1.206;
   1:L PR[91] R[100]mm/sec CNT100;
   1:  PR[91,1] = PR[90,1] + -10.585;
   1:  PR[91,2] = PR[90,2] + -13.526;
   1:  PR[91,3] = PR[90,3] + 1.211;
   1:L PR[91] R[100]mm/sec CNT100;
   1:  PR[91,1] = PR[90,1] + -9.685;
   1:  PR[91,2] = PR[90,2] + -12.864;
   1:  PR[91,3] = PR[90,3] + 1.218;
   1:L PR[91] R[100]mm/sec CNT100;
   1:  PR[91,1] = PR[90,1] + -8.744;
   1:  PR[91,2] = PR[90,2] + -12.069;
   1:  PR[91,3] = PR[90,3] + 1.225;
   1:L PR[91] R[100]mm/sec CNT100;
   1:  PR[91,1] = PR[90,1] + -8.311;
   1:  PR[91,2] = PR[90,2] + -11.662;
   1:  PR[91,3] = PR[90,3] + 1.232;
   1:L PR[91] R[100]mm/sec CNT100;
   1:  PR[91,1] = PR[90,1] + -7.808;
   1:  PR[91,2] = PR[90,2] + -11.150;
   1:  PR[91,3] = PR[90,3] + 1.236;
   1:L PR[91] R[100]mm/sec CNT100;
   1:  PR[91,1] = PR[90,1] + -7.067;
   1:  PR[91,2] = PR[90,2] + -10.304;
   1:  PR[91,3] = PR[90,3] + 1.240;
   1:L PR[91] R[100]mm/sec CNT100;
   1:  PR[91,1] = PR[90,1] + -6.322;
   1:  PR[91,2] = PR[90,2] + -9.329;
   1:  PR[91,3] = PR[90,3] + 1.247;
   1:L PR[91] R[100]mm/sec CNT100;
   1:  PR[91,1] = PR[90,1] + -5.942;
   1:  PR[91,2] = PR[90,2] + -8.770;
   1:  PR[91,3] = PR[90,3] + 1.255;
   1:L PR[91] R[100]mm/sec CNT100;
   1:  PR[91,1] = PR[90,1] + -5.604;
   1:  PR[91,2] = PR[90,2] + -8.228;
   1:  PR[91,3] = PR[90,3] + 1.259;
   1:L PR[91] R[100]mm/sec CNT100;
   1:  PR[91,1] = PR[90,1] + -5.015;
   1:  PR[91,2] = PR[90,2] + -7.153;
   1:  PR[91,3] = PR[90,3] + 1.263;
   1:L PR[91] R[100]mm/sec CNT100;
   1:  PR[91,1] = PR[90,1] + -4.506;
   1:  PR[91,2] = PR[90,2] + -6.040;
   1:  PR[91,3] = PR[90,3] + 1.270;
   1:L PR[91] R[100]mm/sec CNT100;
   1:  PR[91,1] = PR[90,1] + -4.080;
   1:  PR[91,2] = PR[90,2] + -4.896;
   1:  PR[91,3] = PR[90,3] + 1.278;
   1:L PR[91] R[100]mm/sec CNT100;
   1:  PR[91,1] = PR[90,1] + -3.737;
   1:  PR[91,2] = PR[90,2] + -3.722;
   1:  PR[91,3] = PR[90,3] + 1.285;
   1:L PR[91] R[100]mm/sec CNT100;
   1:  PR[91,1] = PR[90,1] + -3.570;
   1:  PR[91,2] = PR[90,2] + -2.996;
   1:  PR[91,3] = PR[90,3] + 1.292;
   1:L PR[91] R[100]mm/sec CNT100;
   1:  PR[91,1] = PR[90,1] + -3.474;
   1:  PR[91,2] = PR[90,2] + -2.500;
   1:  PR[91,3] = PR[90,3] + 1.297;
   1:L PR[91] R[100]mm/sec CNT100;
   1:  PR[91,1] = PR[90,1] + -3.343;
   1:  PR[91,2] = PR[90,2] + -2.011;
   1:  PR[91,3] = PR[90,3] + 1.300;
   1:L PR[91] R[100]mm/sec CNT100;
   1:  PR[91,1] = PR[90,1] + -3.114;
   1:  PR[91,2] = PR[90,2] + -1.522;
   1:  PR[91,3] = PR[90,3] + 1.303;
   1:L PR[91] R[100]mm/sec CNT100;
   1:  PR[91,1] = PR[90,1] + -2.828;
   1:  PR[91,2] = PR[90,2] + -1.108;
   1:  PR[91,3] = PR[90,3] + 1.306;
   1:L PR[91] R[100]mm/sec CNT100;
   1:  PR[91,1] = PR[90,1] + -2.424;
   1:  PR[91,2] = PR[90,2] + -0.697;
   1:  PR[91,3] = PR[90,3] + 1.309;
   1:L PR[91] R[100]mm/sec CNT100;
   1:  PR[91,1] = PR[90,1] + -2.010;
   1:  PR[91,2] = PR[90,2] + -0.405;
   1:  PR[91,3] = PR[90,3] + 1.313;
   1:L PR[91] R[100]mm/sec CNT100;
   1:  PR[91,1] = PR[90,1] + -1.450;
   1:  PR[91,2] = PR[90,2] + -0.145;
   1:  PR[91,3] = PR[90,3] + 1.316;
   1:L PR[91] R[100]mm/sec CNT100;
   1:  PR[91,1] = PR[90,1] + -0.963;
   1:  PR[91,2] = PR[90,2] + -0.016;
   1:  PR[91,3] = PR[90,3] + 1.320;
   1:L PR[91] R[100]mm/sec CNT100;
   1:  PR[91,1] = PR[90,1] + -0.492;
   1:  PR[91,2] = PR[90,2] + 0.026;
   1:  PR[91,3] = PR[90,3] + 1.323;
   1:L PR[91] R[100]mm/sec CNT100;
   1:  PR[91,1] = PR[90,1] + 0.213;
   1:  PR[91,2] = PR[90,2] + 0.028;
   1:  PR[91,3] = PR[90,3] + 1.326;
   1:L PR[91] R[100]mm/sec CNT100;
   1:  PR[91] = PR[90];
   1:  PR[91,1] = PR[90,1] + 0.574;
   1:  PR[91,2] = PR[90,2] + 0.002;
   1:  PR[91,3] = PR[90,3] + 2.660;
   1:L PR[91] R[100]mm/sec CNT100;
   1:  PR[91,1] = PR[90,1] + 0.738;
   1:  PR[91,2] = PR[90,2] + -0.020;
   1:  PR[91,3] = PR[90,3] + 1.332;
   1:L PR[91] R[100]mm/sec CNT100;
   1:  PR[91,1] = PR[90,1] + 1.244;
   1:  PR[91,2] = PR[90,2] + -0.156;
   1:  PR[91,3] = PR[90,3] + 1.333;
   1:L PR[91] R[100]mm/sec CNT100;
   1:  PR[91,1] = PR[90,1] + 1.615;
   1:  PR[91,2] = PR[90,2] + -0.322;
   1:  PR[91,3] = PR[90,3] + 1.336;
   1:L PR[91] R[100]mm/sec CNT100;
   1:  PR[91,1] = PR[90,1] + 1.857;
   1:  PR[91,2] = PR[90,2] + -0.461;
   1:  PR[91,3] = PR[90,3] + 1.339;
   1:L PR[91] R[100]mm/sec CNT100;
   1:  PR[91,1] = PR[90,1] + 2.182;
   1:  PR[91,2] = PR[90,2] + -0.695;
   1:  PR[91,3] = PR[90,3] + 1.341;
   1:L PR[91] R[100]mm/sec CNT100;
   1:  PR[91,1] = PR[90,1] + 2.460;
   1:  PR[91,2] = PR[90,2] + -0.965;
   1:  PR[91,3] = PR[90,3] + 1.343;
   1:L PR[91] R[100]mm/sec CNT100;
   1:  PR[91,1] = PR[90,1] + 2.572;
   1:  PR[91,2] = PR[90,2] + -1.087;
   1:  PR[91,3] = PR[90,3] + 1.345;
   1:L PR[91] R[100]mm/sec CNT100;
   1:  PR[91,1] = PR[90,1] + 2.872;
   1:  PR[91,2] = PR[90,2] + -1.516;
   1:  PR[91,3] = PR[90,3] + 1.346;
   1:L PR[91] R[100]mm/sec CNT100;
   1:  PR[91,1] = PR[90,1] + 3.050;
   1:  PR[91,2] = PR[90,2] + -1.881;
   1:  PR[91,3] = PR[90,3] + 1.350;
   1:L PR[91] R[100]mm/sec CNT100;
   1:  PR[91,1] = PR[90,1] + 3.148;
   1:  PR[91,2] = PR[90,2] + -2.151;
   1:  PR[91,3] = PR[90,3] + 1.352;
   1:L PR[91] R[100]mm/sec CNT100;
   1:  PR[91,1] = PR[90,1] + 3.499;
   1:  PR[91,2] = PR[90,2] + -3.725;
   1:  PR[91,3] = PR[90,3] + 1.354;
   1:L PR[91] R[100]mm/sec CNT100;
   1:  PR[91,1] = PR[90,1] + 3.753;
   1:  PR[91,2] = PR[90,2] + -4.613;
   1:  PR[91,3] = PR[90,3] + 1.364;
   1:L PR[91] R[100]mm/sec CNT100;
   1:  PR[91,1] = PR[90,1] + 3.840;
   1:  PR[91,2] = PR[90,2] + -4.892;
   1:  PR[91,3] = PR[90,3] + 1.369;
   1:L PR[91] R[100]mm/sec CNT100;
   1:  PR[91,1] = PR[90,1] + 4.268;
   1:  PR[91,2] = PR[90,2] + -6.041;
   1:  PR[91,3] = PR[90,3] + 1.371;
   1:L PR[91] R[100]mm/sec CNT100;
   1:  PR[91,1] = PR[90,1] + 4.778;
   1:  PR[91,2] = PR[90,2] + -7.155;
   1:  PR[91,3] = PR[90,3] + 1.378;
   1:L PR[91] R[100]mm/sec CNT100;
   1:  PR[91,1] = PR[90,1] + 5.212;
   1:  PR[91,2] = PR[90,2] + -7.960;
   1:  PR[91,3] = PR[90,3] + 1.386;
   1:L PR[91] R[100]mm/sec CNT100;
   1:  PR[91,1] = PR[90,1] + 5.699;
   1:  PR[91,2] = PR[90,2] + -8.764;
   1:  PR[91,3] = PR[90,3] + 1.391;
   1:L PR[91] R[100]mm/sec CNT100;
   1:  PR[91,1] = PR[90,1] + 6.024;
   1:  PR[91,2] = PR[90,2] + -9.247;
   1:  PR[91,3] = PR[90,3] + 1.397;
   1:L PR[91] R[100]mm/sec CNT100;
   1:  PR[91,1] = PR[90,1] + 6.763;
   1:  PR[91,2] = PR[90,2] + -10.227;
   1:  PR[91,3] = PR[90,3] + 1.401;
   1:L PR[91] R[100]mm/sec CNT100;
   1:  PR[91,1] = PR[90,1] + 7.571;
   1:  PR[91,2] = PR[90,2] + -11.151;
   1:  PR[91,3] = PR[90,3] + 1.408;
   1:L PR[91] R[100]mm/sec CNT100;
   1:  PR[91,1] = PR[90,1] + 8.042;
   1:  PR[91,2] = PR[90,2] + -11.633;
   1:  PR[91,3] = PR[90,3] + 1.416;
   1:L PR[91] R[100]mm/sec CNT100;
   1:  PR[91,1] = PR[90,1] + 8.431;
   1:  PR[91,2] = PR[90,2] + -12.003;
   1:  PR[91,3] = PR[90,3] + 1.420;
   1:L PR[91] R[100]mm/sec CNT100;
   1:  PR[91,1] = PR[90,1] + 9.365;
   1:  PR[91,2] = PR[90,2] + -12.802;
   1:  PR[91,3] = PR[90,3] + 1.423;
   1:L PR[91] R[100]mm/sec CNT100;
   1:  PR[91,1] = PR[90,1] + 10.348;
   1:  PR[91,2] = PR[90,2] + -13.527;
   1:  PR[91,3] = PR[90,3] + 1.430;
   1:L PR[91] R[100]mm/sec CNT100;
   1:  PR[91,1] = PR[90,1] + 11.385;
   1:  PR[91,2] = PR[90,2] + -14.182;
   1:  PR[91,3] = PR[90,3] + 1.438;
   1:L PR[91] R[100]mm/sec CNT100;
   1:  PR[91,1] = PR[90,1] + 12.014;
   1:  PR[91,2] = PR[90,2] + -14.529;
   1:  PR[91,3] = PR[90,3] + 1.445;
   1:L PR[91] R[100]mm/sec CNT100;
   1:  PR[91,1] = PR[90,1] + 12.454;
   1:  PR[91,2] = PR[90,2] + -14.753;
   1:  PR[91,3] = PR[90,3] + 1.450;
   1:L PR[91] R[100]mm/sec CNT100;
   1:  PR[91,1] = PR[90,1] + 13.576;
   1:  PR[91,2] = PR[90,2] + -15.252;
   1:  PR[91,3] = PR[90,3] + 1.453;
   1:L PR[91] R[100]mm/sec CNT100;
   1:  PR[91,1] = PR[90,1] + 14.726;
   1:  PR[91,2] = PR[90,2] + -15.667;
   1:  PR[91,3] = PR[90,3] + 1.460;
   1:L PR[91] R[100]mm/sec CNT100;
   1:  PR[91,1] = PR[90,1] + 15.904;
   1:  PR[91,2] = PR[90,2] + -15.997;
   1:  PR[91,3] = PR[90,3] + 1.467;
   1:L PR[91] R[100]mm/sec CNT100;
   1:  PR[91,1] = PR[90,1] + 16.808;
   1:  PR[91,2] = PR[90,2] + -16.188;
   1:  PR[91,3] = PR[90,3] + 1.475;
   1:L PR[91] R[100]mm/sec CNT100;
   1:  PR[91,1] = PR[90,1] + 17.095;
   1:  PR[91,2] = PR[90,2] + -16.241;
   1:  PR[91,3] = PR[90,3] + 1.481;
   1:L PR[91] R[100]mm/sec CNT100;
   1:  PR[91,1] = PR[90,1] + 18.311;
   1:  PR[91,2] = PR[90,2] + -16.399;
   1:  PR[91,3] = PR[90,3] + 1.482;
   1:L PR[91] R[100]mm/sec CNT100;
   1:  PR[91,1] = PR[90,1] + 19.532;
   1:  PR[91,2] = PR[90,2] + -16.468;
   1:  PR[91,3] = PR[90,3] + 1.490;
   1:L PR[91] R[100]mm/sec CNT100;
   1:  PR[91,1] = PR[90,1] + 20.755;
   1:  PR[91,2] = PR[90,2] + -16.449;
   1:  PR[91,3] = PR[90,3] + 1.497;
   1:L PR[91] R[100]mm/sec CNT100;
   1:  PR[91,1] = PR[90,1] + 21.676;
   1:  PR[91,2] = PR[90,2] + -16.374;
   1:  PR[91,3] = PR[90,3] + 1.505;
   1:L PR[91] R[100]mm/sec CNT100;
   1:  PR[91,1] = PR[90,1] + 21.966;
   1:  PR[91,2] = PR[90,2] + -16.343;
   1:  PR[91,3] = PR[90,3] + 1.510;
   1:L PR[91] R[100]mm/sec CNT100;
   1:  PR[91,1] = PR[90,1] + 23.177;
   1:  PR[91,2] = PR[90,2] + -16.147;
   1:  PR[91,3] = PR[90,3] + 1.512;
   1:L PR[91] R[100]mm/sec CNT100;
   1:  PR[91,1] = PR[90,1] + 24.369;
   1:  PR[91,2] = PR[90,2] + -15.865;
   1:  PR[91,3] = PR[90,3] + 1.519;
   1:L PR[91] R[100]mm/sec CNT100;
   1:  PR[91,1] = PR[90,1] + 25.250;
   1:  PR[91,2] = PR[90,2] + -15.594;
   1:  PR[91,3] = PR[90,3] + 1.527;
   1:L PR[91] R[100]mm/sec CNT100;
   1:  PR[91,1] = PR[90,1] + 25.527;
   1:  PR[91,2] = PR[90,2] + -15.501;
   1:  PR[91,3] = PR[90,3] + 1.532;
   1:L PR[91] R[100]mm/sec CNT100;
   1:  PR[91,1] = PR[90,1] + 26.669;
   1:  PR[91,2] = PR[90,2] + -15.049;
   1:  PR[91,3] = PR[90,3] + 1.534;
   1:L PR[91] R[100]mm/sec CNT100;
   1:  PR[91,1] = PR[90,1] + 27.770;
   1:  PR[91,2] = PR[90,2] + -14.518;
   1:  PR[91,3] = PR[90,3] + 1.542;
   1:L PR[91] R[100]mm/sec CNT100;
   1:  PR[91,1] = PR[90,1] + 28.831;
   1:  PR[91,2] = PR[90,2] + -13.907;
   1:  PR[91,3] = PR[90,3] + 1.549;
   1:L PR[91] R[100]mm/sec CNT100;
   1:  PR[91,1] = PR[90,1] + 29.599;
   1:  PR[91,2] = PR[90,2] + -13.395;
   1:  PR[91,3] = PR[90,3] + 1.557;
   1:L PR[91] R[100]mm/sec CNT100;
   1:  PR[91,1] = PR[90,1] + 29.838;
   1:  PR[91,2] = PR[90,2] + -13.227;
   1:  PR[91,3] = PR[90,3] + 1.562;
   1:L PR[91] R[100]mm/sec CNT100;
   1:  PR[91,1] = PR[90,1] + 30.802;
   1:  PR[91,2] = PR[90,2] + -12.469;
   1:  PR[91,3] = PR[90,3] + 1.564;
   1:L PR[91] R[100]mm/sec CNT100;
   1:  PR[91,1] = PR[90,1] + 31.706;
   1:  PR[91,2] = PR[90,2] + -11.645;
   1:  PR[91,3] = PR[90,3] + 1.571;
   1:L PR[91] R[100]mm/sec CNT100;
   1:  PR[91,1] = PR[90,1] + 32.549;
   1:  PR[91,2] = PR[90,2] + -10.758;
   1:  PR[91,3] = PR[90,3] + 1.579;
   1:L PR[91] R[100]mm/sec CNT100;
   1:  PR[91,1] = PR[90,1] + 33.139;
   1:  PR[91,2] = PR[90,2] + -10.048;
   1:  PR[91,3] = PR[90,3] + 1.586;
   1:L PR[91] R[100]mm/sec CNT100;
   1:  PR[91,1] = PR[90,1] + 33.320;
   1:  PR[91,2] = PR[90,2] + -9.819;
   1:  PR[91,3] = PR[90,3] + 1.592;
   1:L PR[91] R[100]mm/sec CNT100;
   1:  PR[91,1] = PR[90,1] + 34.044;
   1:  PR[91,2] = PR[90,2] + -8.792;
   1:  PR[91,3] = PR[90,3] + 1.594;
   1:L PR[91] R[100]mm/sec CNT100;
   1:  PR[91,1] = PR[90,1] + 34.660;
   1:  PR[91,2] = PR[90,2] + -7.769;
   1:  PR[91,3] = PR[90,3] + 1.601;
   1:L PR[91] R[100]mm/sec CNT100;
   1:  PR[91,1] = PR[90,1] + 35.215;
   1:  PR[91,2] = PR[90,2] + -6.677;
   1:  PR[91,3] = PR[90,3] + 1.609;
   1:L PR[91] R[100]mm/sec CNT100;
   1:  PR[91,1] = PR[90,1] + 35.512;
   1:  PR[91,2] = PR[90,2] + -5.994;
   1:  PR[91,3] = PR[90,3] + 1.616;
   1:L PR[91] R[100]mm/sec CNT100;
   1:  PR[91,1] = PR[90,1] + 35.685;
   1:  PR[91,2] = PR[90,2] + -5.558;
   1:  PR[91,3] = PR[90,3] + 1.621;
   1:L PR[91] R[100]mm/sec CNT100;
   1:  PR[91,1] = PR[90,1] + 36.078;
   1:  PR[91,2] = PR[90,2] + -4.394;
   1:  PR[91,3] = PR[90,3] + 1.623;
   1:L PR[91] R[100]mm/sec CNT100;
   1:  PR[91,1] = PR[90,1] + 36.313;
   1:  PR[91,2] = PR[90,2] + -3.506;
   1:  PR[91,3] = PR[90,3] + 1.631;
   1:L PR[91] R[100]mm/sec CNT100;
   1:  PR[91,1] = PR[90,1] + 36.470;
   1:  PR[91,2] = PR[90,2] + -2.791;
   1:  PR[91,3] = PR[90,3] + 1.636;
   1:L PR[91] R[100]mm/sec CNT100;
   1:  PR[91,1] = PR[90,1] + 36.604;
   1:  PR[91,2] = PR[90,2] + -2.011;
   1:  PR[91,3] = PR[90,3] + 1.641;
   1:L PR[91] R[100]mm/sec CNT100;
   1:  PR[91,1] = PR[90,1] + 36.708;
   1:  PR[91,2] = PR[90,2] + -1.100;
   1:  PR[91,3] = PR[90,3] + 1.646;
   1:L PR[91] R[100]mm/sec CNT100;
   1:  PR[91,1] = PR[90,1] + 36.771;
   1:  PR[91,2] = PR[90,2] + -0.122;
   1:  PR[91,3] = PR[90,3] + 1.651;
   1:L PR[91] R[100]mm/sec CNT100;
   1:  PR[91,1] = PR[90,1] + 36.781;
   1:  PR[91,2] = PR[90,2] + 0.423;
   1:  PR[91,3] = PR[90,3] + 1.657;
   1:L PR[91] R[100]mm/sec CNT100;
   1:  PR[91,1] = PR[90,1] + 36.752;
   1:  PR[91,2] = PR[90,2] + 1.349;
   1:  PR[91,3] = PR[90,3] + 1.660;
   1:L PR[91] R[100]mm/sec CNT100;
   1:  PR[91,1] = PR[90,1] + 36.709;
   1:  PR[91,2] = PR[90,2] + 1.953;
   1:  PR[91,3] = PR[90,3] + 1.666;
   1:L PR[91] R[100]mm/sec CNT100;
   1:  PR[91,1] = PR[90,1] + 36.604;
   1:  PR[91,2] = PR[90,2] + 2.865;
   1:  PR[91,3] = PR[90,3] + 1.670;
   1:L PR[91] R[100]mm/sec CNT100;
   1:  PR[91,1] = PR[90,1] + 36.444;
   1:  PR[91,2] = PR[90,2] + 3.769;
   1:  PR[91,3] = PR[90,3] + 1.675;
   1:L PR[91] R[100]mm/sec CNT100;
   1:  PR[91,1] = PR[90,1] + 36.313;
   1:  PR[91,2] = PR[90,2] + 4.361;
   1:  PR[91,3] = PR[90,3] + 1.681;
   1:L PR[91] R[100]mm/sec CNT100;
   1:  PR[91,1] = PR[90,1] + 36.077;
   1:  PR[91,2] = PR[90,2] + 5.255;
   1:  PR[91,3] = PR[90,3] + 1.685;
   1:L PR[91] R[100]mm/sec CNT100;
   1:  PR[91,1] = PR[90,1] + 35.911;
   1:  PR[91,2] = PR[90,2] + 5.778;
   1:  PR[91,3] = PR[90,3] + 1.690;
   1:L PR[91] R[100]mm/sec CNT100;
   1:  PR[91,1] = PR[90,1] + 35.574;
   1:  PR[91,2] = PR[90,2] + 6.691;
   1:  PR[91,3] = PR[90,3] + 1.694;
   1:L PR[91] R[100]mm/sec CNT100;
   1:  PR[91,1] = PR[90,1] + 35.213;
   1:  PR[91,2] = PR[90,2] + 7.535;
   1:  PR[91,3] = PR[90,3] + 1.699;
   1:L PR[91] R[100]mm/sec CNT100;
   1:  PR[91,1] = PR[90,1] + 34.800;
   1:  PR[91,2] = PR[90,2] + 8.359;
   1:  PR[91,3] = PR[90,3] + 1.705;
   1:L PR[91] R[100]mm/sec CNT100;
   1:  PR[91,1] = PR[90,1] + 34.506;
   1:  PR[91,2] = PR[90,2] + 8.889;
   1:  PR[91,3] = PR[90,3] + 1.711;
   1:L PR[91] R[100]mm/sec CNT100;
   1:  PR[91,1] = PR[90,1] + 34.028;
   1:  PR[91,2] = PR[90,2] + 9.672;
   1:  PR[91,3] = PR[90,3] + 1.714;
   1:L PR[91] R[100]mm/sec CNT100;
   1:  PR[91,1] = PR[90,1] + 33.503;
   1:  PR[91,2] = PR[90,2] + 10.425;
   1:  PR[91,3] = PR[90,3] + 1.720;
   1:L PR[91] R[100]mm/sec CNT100;
   1:  PR[91,1] = PR[90,1] + 33.136;
   1:  PR[91,2] = PR[90,2] + 10.907;
   1:  PR[91,3] = PR[90,3] + 1.725;
   1:L PR[91] R[100]mm/sec CNT100;
   1:  PR[91,1] = PR[90,1] + 32.548;
   1:  PR[91,2] = PR[90,2] + 11.614;
   1:  PR[91,3] = PR[90,3] + 1.729;
   1:L PR[91] R[100]mm/sec CNT100;
   1:  PR[91,1] = PR[90,1] + 31.919;
   1:  PR[91,2] = PR[90,2] + 12.285;
   1:  PR[91,3] = PR[90,3] + 1.735;
   1:L PR[91] R[100]mm/sec CNT100;
   1:  PR[91,1] = PR[90,1] + 31.486;
   1:  PR[91,2] = PR[90,2] + 12.708;
   1:  PR[91,3] = PR[90,3] + 1.740;
   1:L PR[91] R[100]mm/sec CNT100;
   1:  PR[91,1] = PR[90,1] + 30.804;
   1:  PR[91,2] = PR[90,2] + 13.323;
   1:  PR[91,3] = PR[90,3] + 1.744;
   1:L PR[91] R[100]mm/sec CNT100;
   1:  PR[91,1] = PR[90,1] + 29.838;
   1:  PR[91,2] = PR[90,2] + 14.083;
   1:  PR[91,3] = PR[90,3] + 1.750;
   1:L PR[91] R[100]mm/sec CNT100;
   1:  PR[91,1] = PR[90,1] + 29.336;
   1:  PR[91,2] = PR[90,2] + 14.435;
   1:  PR[91,3] = PR[90,3] + 1.757;
   1:L PR[91] R[100]mm/sec CNT100;
   1:  PR[91,1] = PR[90,1] + 28.833;
   1:  PR[91,2] = PR[90,2] + 14.762;
   1:  PR[91,3] = PR[90,3] + 1.761;
   1:L PR[91] R[100]mm/sec CNT100;
   1:  PR[91,1] = PR[90,1] + 28.035;
   1:  PR[91,2] = PR[90,2] + 15.227;
   1:  PR[91,3] = PR[90,3] + 1.764;
   1:L PR[91] R[100]mm/sec CNT100;
   1:  PR[91,1] = PR[90,1] + 27.499;
   1:  PR[91,2] = PR[90,2] + 15.510;
   1:  PR[91,3] = PR[90,3] + 1.770;
   1:L PR[91] R[100]mm/sec CNT100;
   1:  PR[91,1] = PR[90,1] + 26.669;
   1:  PR[91,2] = PR[90,2] + 15.904;
   1:  PR[91,3] = PR[90,3] + 1.774;
   1:L PR[91] R[100]mm/sec CNT100;
   1:  PR[91,1] = PR[90,1] + 25.816;
   1:  PR[91,2] = PR[90,2] + 16.248;
   1:  PR[91,3] = PR[90,3] + 1.779;
   1:L PR[91] R[100]mm/sec CNT100;
   1:  PR[91,1] = PR[90,1] + 25.245;
   1:  PR[91,2] = PR[90,2] + 16.450;
   1:  PR[91,3] = PR[90,3] + 1.785;
   1:L PR[91] R[100]mm/sec CNT100;
   1:  PR[91,1] = PR[90,1] + 24.369;
   1:  PR[91,2] = PR[90,2] + 16.720;
   1:  PR[91,3] = PR[90,3] + 1.789;
   1:L PR[91] R[100]mm/sec CNT100;
   1:  PR[91,1] = PR[90,1] + 23.175;
   1:  PR[91,2] = PR[90,2] + 17.003;
   1:  PR[91,3] = PR[90,3] + 1.794;
   1:L PR[91] R[100]mm/sec CNT100;
   1:  PR[91,1] = PR[90,1] + 22.272;
   1:  PR[91,2] = PR[90,2] + 17.154;
   1:  PR[91,3] = PR[90,3] + 1.802;
   1:L PR[91] R[100]mm/sec CNT100;
   1:  PR[91,1] = PR[90,1] + 21.670;
   1:  PR[91,2] = PR[90,2] + 17.229;
   1:  PR[91,3] = PR[90,3] + 1.807;
   1:L PR[91] R[100]mm/sec CNT100;
   1:  PR[91,1] = PR[90,1] + 20.750;
   1:  PR[91,2] = PR[90,2] + 17.305;
   1:  PR[91,3] = PR[90,3] + 1.811;
   1:L PR[91] R[100]mm/sec CNT100;
   1:  PR[91,1] = PR[90,1] + 20.456;
   1:  PR[91,2] = PR[90,2] + 17.315;
   1:  PR[91,3] = PR[90,3] + 1.816;
   1:L PR[91] R[100]mm/sec CNT100;
   1:  PR[91,1] = PR[90,1] + 19.532;
   1:  PR[91,2] = PR[90,2] + 17.324;
   1:  PR[91,3] = PR[90,3] + 1.818;
   1:L PR[91] R[100]mm/sec CNT100;
   1:  PR[91,1] = PR[90,1] + 18.613;
   1:  PR[91,2] = PR[90,2] + 17.277;
   1:  PR[91,3] = PR[90,3] + 1.824;
   1:L PR[91] R[100]mm/sec CNT100;
   1:  PR[91,1] = PR[90,1] + 18.010;
   1:  PR[91,2] = PR[90,2] + 17.221;
   1:  PR[91,3] = PR[90,3] + 1.829;
   1:L PR[91] R[100]mm/sec CNT100;
   1:  PR[91,1] = PR[90,1] + 17.102;
   1:  PR[91,2] = PR[90,2] + 17.097;
   1:  PR[91,3] = PR[90,3] + 1.833;
   1:L PR[91] R[100]mm/sec CNT100;
   1:  PR[91,1] = PR[90,1] + 15.902;
   1:  PR[91,2] = PR[90,2] + 16.852;
   1:  PR[91,3] = PR[90,3] + 1.839;
   1:L PR[91] R[100]mm/sec CNT100;
   1:  PR[91,1] = PR[90,1] + 14.726;
   1:  PR[91,2] = PR[90,2] + 16.522;
   1:  PR[91,3] = PR[90,3] + 1.846;
   1:L PR[91] R[100]mm/sec CNT100;
   1:  PR[91,1] = PR[90,1] + 13.576;
   1:  PR[91,2] = PR[90,2] + 16.107;
   1:  PR[91,3] = PR[90,3] + 1.854;
   1:L PR[91] R[100]mm/sec CNT100;
   1:  PR[91,1] = PR[90,1] + 12.459;
   1:  PR[91,2] = PR[90,2] + 15.610;
   1:  PR[91,3] = PR[90,3] + 1.861;
   1:L PR[91] R[100]mm/sec CNT100;
   1:  PR[91,1] = PR[90,1] + 11.382;
   1:  PR[91,2] = PR[90,2] + 15.034;
   1:  PR[91,3] = PR[90,3] + 1.868;
   1:L PR[91] R[100]mm/sec CNT100;
   1:  PR[91,1] = PR[90,1] + 10.346;
   1:  PR[91,2] = PR[90,2] + 14.381;
   1:  PR[91,3] = PR[90,3] + 1.876;
   1:L PR[91] R[100]mm/sec CNT100;
   1:  PR[91,1] = PR[90,1] + 9.605;
   1:  PR[91,2] = PR[90,2] + 13.841;
   1:  PR[91,3] = PR[90,3] + 1.883;
   1:L PR[91] R[100]mm/sec CNT100;
   1:  PR[91,1] = PR[90,1] + 9.131;
   1:  PR[91,2] = PR[90,2] + 13.464;
   1:  PR[91,3] = PR[90,3] + 1.889;
   1:L PR[91] R[100]mm/sec CNT100;
   1:  PR[91,1] = PR[90,1] + 8.436;
   1:  PR[91,2] = PR[90,2] + 12.862;
   1:  PR[91,3] = PR[90,3] + 1.892;
   1:L PR[91] R[100]mm/sec CNT100;
   1:  PR[91,1] = PR[90,1] + 7.780;
   1:  PR[91,2] = PR[90,2] + 12.221;
   1:  PR[91,3] = PR[90,3] + 1.898;
   1:L PR[91] R[100]mm/sec CNT100;
   1:  PR[91,1] = PR[90,1] + 7.150;
   1:  PR[91,2] = PR[90,2] + 11.541;
   1:  PR[91,3] = PR[90,3] + 1.904;
   1:L PR[91] R[100]mm/sec CNT100;
   1:  PR[91,1] = PR[90,1] + 6.766;
   1:  PR[91,2] = PR[90,2] + 11.086;
   1:  PR[91,3] = PR[90,3] + 1.909;
   1:L PR[91] R[100]mm/sec CNT100;
   1:  PR[91,1] = PR[90,1] + 6.027;
   1:  PR[91,2] = PR[90,2] + 10.105;
   1:  PR[91,3] = PR[90,3] + 1.913;
   1:L PR[91] R[100]mm/sec CNT100;
   1:  PR[91,1] = PR[90,1] + 5.524;
   1:  PR[91,2] = PR[90,2] + 9.338;
   1:  PR[91,3] = PR[90,3] + 1.920;
   1:L PR[91] R[100]mm/sec CNT100;
   1:  PR[91,1] = PR[90,1] + 5.085;
   1:  PR[91,2] = PR[90,2] + 8.593;
   1:  PR[91,3] = PR[90,3] + 1.926;
   1:L PR[91] R[100]mm/sec CNT100;
   1:  PR[91,1] = PR[90,1] + 4.645;
   1:  PR[91,2] = PR[90,2] + 7.733;
   1:  PR[91,3] = PR[90,3] + 1.931;
   1:L PR[91] R[100]mm/sec CNT100;
   1:  PR[91,1] = PR[90,1] + 4.267;
   1:  PR[91,2] = PR[90,2] + 6.893;
   1:  PR[91,3] = PR[90,3] + 1.937;
   1:L PR[91] R[100]mm/sec CNT100;
   1:  PR[91,1] = PR[90,1] + 4.159;
   1:  PR[91,2] = PR[90,2] + 6.620;
   1:  PR[91,3] = PR[90,3] + 1.943;
   1:L PR[91] R[100]mm/sec CNT100;
   1:  PR[91,1] = PR[90,1] + 3.838;
   1:  PR[91,2] = PR[90,2] + 5.742;
   1:  PR[91,3] = PR[90,3] + 1.944;
   1:L PR[91] R[100]mm/sec CNT100;
   1:  PR[91,1] = PR[90,1] + 3.579;
   1:  PR[91,2] = PR[90,2] + 4.873;
   1:  PR[91,3] = PR[90,3] + 1.950;
   1:L PR[91] R[100]mm/sec CNT100;
   1:  PR[91,1] = PR[90,1] + 3.430;
   1:  PR[91,2] = PR[90,2] + 4.286;
   1:  PR[91,3] = PR[90,3] + 1.956;
   1:L PR[91] R[100]mm/sec CNT100;
   1:  PR[91,1] = PR[90,1] + 3.234;
   1:  PR[91,2] = PR[90,2] + 3.349;
   1:  PR[91,3] = PR[90,3] + 1.959;
   1:L PR[91] R[100]mm/sec CNT100;
   1:  PR[91,1] = PR[90,1] + 3.104;
   1:  PR[91,2] = PR[90,2] + 2.865;
   1:  PR[91,3] = PR[90,3] + 1.965;
   1:L PR[91] R[100]mm/sec CNT100;
   1:  PR[91,1] = PR[90,1] + 2.875;
   1:  PR[91,2] = PR[90,2] + 2.375;
   1:  PR[91,3] = PR[90,3] + 1.968;
   1:L PR[91] R[100]mm/sec CNT100;
   1:  PR[91,1] = PR[90,1] + 2.564;
   1:  PR[91,2] = PR[90,2] + 1.931;
   1:  PR[91,3] = PR[90,3] + 1.971;
   1:L PR[91] R[100]mm/sec CNT100;
   1:  PR[91,1] = PR[90,1] + 2.185;
   1:  PR[91,2] = PR[90,2] + 1.553;
   1:  PR[91,3] = PR[90,3] + 1.975;
   1:L PR[91] R[100]mm/sec CNT100;
   1:  PR[91,1] = PR[90,1] + 1.846;
   1:  PR[91,2] = PR[90,2] + 1.308;
   1:  PR[91,3] = PR[90,3] + 1.978;
   1:L PR[91] R[100]mm/sec CNT100;
   1:  PR[91,1] = PR[90,1] + 1.384;
   1:  PR[91,2] = PR[90,2] + 1.069;
   1:  PR[91,3] = PR[90,3] + 1.981;
   1:L PR[91] R[100]mm/sec CNT100;
   1:  PR[91,1] = PR[90,1] + 1.115;
   1:  PR[91,2] = PR[90,2] + 0.971;
   1:  PR[91,3] = PR[90,3] + 1.984;
   1:L PR[91] R[100]mm/sec CNT100;
   1:  PR[91,1] = PR[90,1] + 0.725;
   1:  PR[91,2] = PR[90,2] + 0.872;
   1:  PR[91,3] = PR[90,3] + 1.985;
   1:L PR[91] R[100]mm/sec CNT100;
   1:  PR[91,1] = PR[90,1] + 0.330;
   1:  PR[91,2] = PR[90,2] + 0.832;
   1:  PR[91,3] = PR[90,3] + 1.988;
   1:L PR[91] R[100]mm/sec CNT100;
   1:  PR[91,1] = PR[90,1] + -0.452;
   1:  PR[91,2] = PR[90,2] + 0.827;
   1:  PR[91,3] = PR[90,3] + 1.990;
   1:L PR[91] R[100]mm/sec CNT100;
   1:  PR[91,1] = PR[90,1] + -0.964;
   1:  PR[91,2] = PR[90,2] + 0.872;
   1:  PR[91,3] = PR[90,3] + 1.995;
   1:L PR[91] R[100]mm/sec CNT100;
   1:  PR[91,1] = PR[90,1] + -1.482;
   1:  PR[91,2] = PR[90,2] + 1.011;
   1:  PR[91,3] = PR[90,3] + 1.998;
   1:L PR[91] R[100]mm/sec CNT100;
   1:  PR[91,1] = PR[90,1] + -1.854;
   1:  PR[91,2] = PR[90,2] + 1.177;
   1:  PR[91,3] = PR[90,3] + 2.001;
   1:L PR[91] R[100]mm/sec CNT100;
   1:  PR[91,1] = PR[90,1] + -2.095;
   1:  PR[91,2] = PR[90,2] + 1.316;
   1:  PR[91,3] = PR[90,3] + 2.004;
   1:L PR[91] R[100]mm/sec CNT100;
   1:  PR[91,1] = PR[90,1] + -2.420;
   1:  PR[91,2] = PR[90,2] + 1.550;
   1:  PR[91,3] = PR[90,3] + 2.006;
   1:L PR[91] R[100]mm/sec CNT100;
   1:  PR[91,1] = PR[90,1] + -2.698;
   1:  PR[91,2] = PR[90,2] + 1.820;
   1:  PR[91,3] = PR[90,3] + 2.008;
   1:L PR[91] R[100]mm/sec CNT100;
   1:  PR[91,1] = PR[90,1] + -2.810;
   1:  PR[91,2] = PR[90,2] + 1.942;
   1:  PR[91,3] = PR[90,3] + 2.010;
   1:L PR[91] R[100]mm/sec CNT100;
   1:  PR[91,1] = PR[90,1] + -3.107;
   1:  PR[91,2] = PR[90,2] + 2.366;
   1:  PR[91,3] = PR[90,3] + 2.011;
   1:L PR[91] R[100]mm/sec CNT100;
   1:  PR[91,1] = PR[90,1] + -3.252;
   1:  PR[91,2] = PR[90,2] + 2.647;
   1:  PR[91,3] = PR[90,3] + 2.015;
   1:L PR[91] R[100]mm/sec CNT100;
   1:  PR[91,1] = PR[90,1] + -3.386;
   1:  PR[91,2] = PR[90,2] + 3.003;
   1:  PR[91,3] = PR[90,3] + 2.016;
   1:L PR[91] R[100]mm/sec CNT100;
   1:  PR[91,1] = PR[90,1] + -3.738;
   1:  PR[91,2] = PR[90,2] + 4.581;
   1:  PR[91,3] = PR[90,3] + 2.019;
   1:L PR[91] R[100]mm/sec CNT100;
   1:  PR[91,1] = PR[90,1] + -3.991;
   1:  PR[91,2] = PR[90,2] + 5.468;
   1:  PR[91,3] = PR[90,3] + 2.029;
   1:L PR[91] R[100]mm/sec CNT100;
   1:  PR[91,1] = PR[90,1] + -4.078;
   1:  PR[91,2] = PR[90,2] + 5.747;
   1:  PR[91,3] = PR[90,3] + 2.034;
   1:L PR[91] R[100]mm/sec CNT100;
   1:  PR[91,1] = PR[90,1] + -4.507;
   1:  PR[91,2] = PR[90,2] + 6.896;
   1:  PR[91,3] = PR[90,3] + 2.036;
   1:L PR[91] R[100]mm/sec CNT100;
   1:  PR[91,1] = PR[90,1] + -5.017;
   1:  PR[91,2] = PR[90,2] + 8.013;
   1:  PR[91,3] = PR[90,3] + 2.043;
   1:L PR[91] R[100]mm/sec CNT100;
   1:  PR[91,1] = PR[90,1] + -5.323;
   1:  PR[91,2] = PR[90,2] + 8.594;
   1:  PR[91,3] = PR[90,3] + 2.051;
   1:L PR[91] R[100]mm/sec CNT100;
   1:  PR[91,1] = PR[90,1] + -5.599;
   1:  PR[91,2] = PR[90,2] + 9.075;
   1:  PR[91,3] = PR[90,3] + 2.055;
   1:L PR[91] R[100]mm/sec CNT100;
   1:  PR[91,1] = PR[90,1] + -6.266;
   1:  PR[91,2] = PR[90,2] + 10.107;
   1:  PR[91,3] = PR[90,3] + 2.058;
   1:L PR[91] R[100]mm/sec CNT100;
   1:  PR[91,1] = PR[90,1] + -7.004;
   1:  PR[91,2] = PR[90,2] + 11.086;
   1:  PR[91,3] = PR[90,3] + 2.066;
   1:L PR[91] R[100]mm/sec CNT100;
   1:  PR[91,1] = PR[90,1] + -7.390;
   1:  PR[91,2] = PR[90,2] + 11.544;
   1:  PR[91,3] = PR[90,3] + 2.073;
   1:L PR[91] R[100]mm/sec CNT100;
   1:  PR[91,1] = PR[90,1] + -7.802;
   1:  PR[91,2] = PR[90,2] + 11.999;
   1:  PR[91,3] = PR[90,3] + 2.077;
   1:L PR[91] R[100]mm/sec CNT100;
   1:  PR[91,1] = PR[90,1] + -8.674;
   1:  PR[91,2] = PR[90,2] + 12.862;
   1:  PR[91,3] = PR[90,3] + 2.080;
   1:L PR[91] R[100]mm/sec CNT100;
   1:  PR[91,1] = PR[90,1] + -9.605;
   1:  PR[91,2] = PR[90,2] + 13.658;
   1:  PR[91,3] = PR[90,3] + 2.088;
   1:L PR[91] R[100]mm/sec CNT100;
   1:  PR[91,1] = PR[90,1] + -10.339;
   1:  PR[91,2] = PR[90,2] + 14.206;
   1:  PR[91,3] = PR[90,3] + 2.095;
   1:L PR[91] R[100]mm/sec CNT100;
   1:  PR[91,1] = PR[90,1] + -10.879;
   1:  PR[91,2] = PR[90,2] + 14.575;
   1:  PR[91,3] = PR[90,3] + 2.101;
   1:L PR[91] R[100]mm/sec CNT100;
   1:  PR[91,1] = PR[90,1] + -11.618;
   1:  PR[91,2] = PR[90,2] + 15.033;
   1:  PR[91,3] = PR[90,3] + 2.105;
   1:L PR[91] R[100]mm/sec CNT100;
   1:  PR[91,1] = PR[90,1] + -12.698;
   1:  PR[91,2] = PR[90,2] + 15.610;
   1:  PR[91,3] = PR[90,3] + 2.110;
   1:L PR[91] R[100]mm/sec CNT100;
   1:  PR[91,1] = PR[90,1] + -13.816;
   1:  PR[91,2] = PR[90,2] + 16.108;
   1:  PR[91,3] = PR[90,3] + 2.118;
   1:L PR[91] R[100]mm/sec CNT100;
   1:  PR[91,1] = PR[90,1] + -14.683;
   1:  PR[91,2] = PR[90,2] + 16.426;
   1:  PR[91,3] = PR[90,3] + 2.125;
   1:L PR[91] R[100]mm/sec CNT100;
   1:  PR[91,1] = PR[90,1] + -14.959;
   1:  PR[91,2] = PR[90,2] + 16.520;
   1:  PR[91,3] = PR[90,3] + 2.131;
   1:L PR[91] R[100]mm/sec CNT100;
   1:  PR[91,1] = PR[90,1] + -16.141;
   1:  PR[91,2] = PR[90,2] + 16.852;
   1:  PR[91,3] = PR[90,3] + 2.132;
   1:L PR[91] R[100]mm/sec CNT100;
   1:  PR[91,1] = PR[90,1] + -17.340;
   1:  PR[91,2] = PR[90,2] + 17.097;
   1:  PR[91,3] = PR[90,3] + 2.140;
   1:L PR[91] R[100]mm/sec CNT100;
   1:  PR[91,1] = PR[90,1] + -18.254;
   1:  PR[91,2] = PR[90,2] + 17.221;
   1:  PR[91,3] = PR[90,3] + 2.147;
   1:L PR[91] R[100]mm/sec CNT100;
   1:  PR[91,1] = PR[90,1] + -18.544;
   1:  PR[91,2] = PR[90,2] + 17.254;
   1:  PR[91,3] = PR[90,3] + 2.153;
   1:L PR[91] R[100]mm/sec CNT100;
   1:  PR[91,1] = PR[90,1] + -19.771;
   1:  PR[91,2] = PR[90,2] + 17.324;
   1:  PR[91,3] = PR[90,3] + 2.155;
   1:L PR[91] R[100]mm/sec CNT100;
   1:  PR[91,1] = PR[90,1] + -20.994;
   1:  PR[91,2] = PR[90,2] + 17.305;
   1:  PR[91,3] = PR[90,3] + 2.162;
   1:L PR[91] R[100]mm/sec CNT100;
   1:  PR[91,1] = PR[90,1] + -21.914;
   1:  PR[91,2] = PR[90,2] + 17.229;
   1:  PR[91,3] = PR[90,3] + 2.170;
   1:L PR[91] R[100]mm/sec CNT100;
   1:  PR[91,1] = PR[90,1] + -22.205;
   1:  PR[91,2] = PR[90,2] + 17.198;
   1:  PR[91,3] = PR[90,3] + 2.175;
   1:L PR[91] R[100]mm/sec CNT100;
   1:  PR[91,1] = PR[90,1] + -23.416;
   1:  PR[91,2] = PR[90,2] + 17.002;
   1:  PR[91,3] = PR[90,3] + 2.177;
   1:L PR[91] R[100]mm/sec CNT100;
   1:  PR[91,1] = PR[90,1] + -24.606;
   1:  PR[91,2] = PR[90,2] + 16.721;
   1:  PR[91,3] = PR[90,3] + 2.184;
   1:L PR[91] R[100]mm/sec CNT100;
   1:  PR[91,1] = PR[90,1] + -25.771;
   1:  PR[91,2] = PR[90,2] + 16.354;
   1:  PR[91,3] = PR[90,3] + 2.192;
   1:L PR[91] R[100]mm/sec CNT100;
   1:  PR[91,1] = PR[90,1] + -26.909;
   1:  PR[91,2] = PR[90,2] + 15.903;
   1:  PR[91,3] = PR[90,3] + 2.199;
   1:L PR[91] R[100]mm/sec CNT100;
   1:  PR[91,1] = PR[90,1] + -27.743;
   1:  PR[91,2] = PR[90,2] + 15.507;
   1:  PR[91,3] = PR[90,3] + 2.207;
   1:L PR[91] R[100]mm/sec CNT100;
   1:  PR[91,1] = PR[90,1] + -28.005;
   1:  PR[91,2] = PR[90,2] + 15.375;
   1:  PR[91,3] = PR[90,3] + 2.212;
   1:L PR[91] R[100]mm/sec CNT100;
   1:  PR[91,1] = PR[90,1] + -28.806;
   1:  PR[91,2] = PR[90,2] + 14.920;
   1:  PR[91,3] = PR[90,3] + 2.214;
   1:L PR[91] R[100]mm/sec CNT100;
   1:  PR[91,1] = PR[90,1] + -29.578;
   1:  PR[91,2] = PR[90,2] + 14.432;
   1:  PR[91,3] = PR[90,3] + 2.220;
   1:L PR[91] R[100]mm/sec CNT100;
   1:  PR[91,1] = PR[90,1] + -30.076;
   1:  PR[91,2] = PR[90,2] + 14.083;
   1:  PR[91,3] = PR[90,3] + 2.225;
   1:L PR[91] R[100]mm/sec CNT100;
   1:  PR[91,1] = PR[90,1] + -31.041;
   1:  PR[91,2] = PR[90,2] + 13.324;
   1:  PR[91,3] = PR[90,3] + 2.229;
   1:L PR[91] R[100]mm/sec CNT100;
   1:  PR[91,1] = PR[90,1] + -31.946;
   1:  PR[91,2] = PR[90,2] + 12.499;
   1:  PR[91,3] = PR[90,3] + 2.236;
   1:L PR[91] R[100]mm/sec CNT100;
   1:  PR[91,1] = PR[90,1] + -32.581;
   1:  PR[91,2] = PR[90,2] + 11.838;
   1:  PR[91,3] = PR[90,3] + 2.244;
   1:L PR[91] R[100]mm/sec CNT100;
   1:  PR[91,1] = PR[90,1] + -33.020;
   1:  PR[91,2] = PR[90,2] + 11.341;
   1:  PR[91,3] = PR[90,3] + 2.249;
   1:L PR[91] R[100]mm/sec CNT100;
   1:  PR[91,1] = PR[90,1] + -33.561;
   1:  PR[91,2] = PR[90,2] + 10.671;
   1:  PR[91,3] = PR[90,3] + 2.253;
   1:L PR[91] R[100]mm/sec CNT100;
   1:  PR[91,1] = PR[90,1] + -34.266;
   1:  PR[91,2] = PR[90,2] + 9.671;
   1:  PR[91,3] = PR[90,3] + 2.259;
   1:L PR[91] R[100]mm/sec CNT100;
   1:  PR[91,1] = PR[90,1] + -34.896;
   1:  PR[91,2] = PR[90,2] + 8.627;
   1:  PR[91,3] = PR[90,3] + 2.266;
   1:L PR[91] R[100]mm/sec CNT100;
   1:  PR[91,1] = PR[90,1] + -35.452;
   1:  PR[91,2] = PR[90,2] + 7.534;
   1:  PR[91,3] = PR[90,3] + 2.274;
   1:L PR[91] R[100]mm/sec CNT100;
   1:  PR[91,1] = PR[90,1] + -35.812;
   1:  PR[91,2] = PR[90,2] + 6.691;
   1:  PR[91,3] = PR[90,3] + 2.281;
   1:L PR[91] R[100]mm/sec CNT100;
   1:  PR[91,1] = PR[90,1] + -36.150;
   1:  PR[91,2] = PR[90,2] + 5.778;
   1:  PR[91,3] = PR[90,3] + 2.287;
   1:L PR[91] R[100]mm/sec CNT100;
   1:  PR[91,1] = PR[90,1] + -36.315;
   1:  PR[91,2] = PR[90,2] + 5.254;
   1:  PR[91,3] = PR[90,3] + 2.292;
   1:L PR[91] R[100]mm/sec CNT100;
   1:  PR[91,1] = PR[90,1] + -36.553;
   1:  PR[91,2] = PR[90,2] + 4.356;
   1:  PR[91,3] = PR[90,3] + 2.296;
   1:L PR[91] R[100]mm/sec CNT100;
   1:  PR[91,1] = PR[90,1] + -36.622;
   1:  PR[91,2] = PR[90,2] + 4.070;
   1:  PR[91,3] = PR[90,3] + 2.301;
   1:L PR[91] R[100]mm/sec CNT100;
   1:  PR[91,1] = PR[90,1] + -36.793;
   1:  PR[91,2] = PR[90,2] + 3.164;
   1:  PR[91,3] = PR[90,3] + 2.303;
   1:L PR[91] R[100]mm/sec CNT100;
   1:  PR[91,1] = PR[90,1] + -36.883;
   1:  PR[91,2] = PR[90,2] + 2.546;
   1:  PR[91,3] = PR[90,3] + 2.309;
   1:L PR[91] R[100]mm/sec CNT100;
   1:  PR[91,1] = PR[90,1] + -36.974;
   1:  PR[91,2] = PR[90,2] + 1.653;
   1:  PR[91,3] = PR[90,3] + 2.313;
   1:L PR[91] R[100]mm/sec CNT100;
   1:  PR[91,1] = PR[90,1] + -37.019;
   1:  PR[91,2] = PR[90,2] + 0.422;
   1:  PR[91,3] = PR[90,3] + 2.318;
   1:L PR[91] R[100]mm/sec CNT100;
   1:  PR[91,1] = PR[90,1] + -37.010;
   1:  PR[91,2] = PR[90,2] + -0.126;
   1:  PR[91,3] = PR[90,3] + 2.326;
   1:L PR[91] R[100]mm/sec CNT100;
   1:  PR[91,1] = PR[90,1] + -36.975;
   1:  PR[91,2] = PR[90,2] + -0.793;
   1:  PR[91,3] = PR[90,3] + 2.329;
   1:L PR[91] R[100]mm/sec CNT100;
   1:  PR[91,1] = PR[90,1] + -36.881;
   1:  PR[91,2] = PR[90,2] + -1.705;
   1:  PR[91,3] = PR[90,3] + 2.333;
   1:L PR[91] R[100]mm/sec CNT100;
   1:  PR[91,1] = PR[90,1] + -36.708;
   1:  PR[91,2] = PR[90,2] + -2.794;
   1:  PR[91,3] = PR[90,3] + 2.338;
   1:L PR[91] R[100]mm/sec CNT100;
   1:  PR[91,1] = PR[90,1] + -36.552;
   1:  PR[91,2] = PR[90,2] + -3.506;
   1:  PR[91,3] = PR[90,3] + 2.345;
   1:L PR[91] R[100]mm/sec CNT100;
   1:  PR[91,1] = PR[90,1] + -36.317;
   1:  PR[91,2] = PR[90,2] + -4.394;
   1:  PR[91,3] = PR[90,3] + 2.350;
   1:L PR[91] R[100]mm/sec CNT100;
   1:  PR[91,1] = PR[90,1] + -35.923;
   1:  PR[91,2] = PR[90,2] + -5.559;
   1:  PR[91,3] = PR[90,3] + 2.355;
   1:L PR[91] R[100]mm/sec CNT100;
   1:  PR[91,1] = PR[90,1] + -35.751;
   1:  PR[91,2] = PR[90,2] + -5.994;
   1:  PR[91,3] = PR[90,3] + 2.363;
   1:L PR[91] R[100]mm/sec CNT100;
   1:  PR[91,1] = PR[90,1] + -35.452;
   1:  PR[91,2] = PR[90,2] + -6.678;
   1:  PR[91,3] = PR[90,3] + 2.366;
   1:L PR[91] R[100]mm/sec CNT100;
   1:  PR[91,1] = PR[90,1] + -35.038;
   1:  PR[91,2] = PR[90,2] + -7.506;
   1:  PR[91,3] = PR[90,3] + 2.370;
   1:L PR[91] R[100]mm/sec CNT100;
   1:  PR[91,1] = PR[90,1] + -34.900;
   1:  PR[91,2] = PR[90,2] + -7.766;
   1:  PR[91,3] = PR[90,3] + 2.376;
   1:L PR[91] R[100]mm/sec CNT100;
   1:  PR[91,1] = PR[90,1] + -34.443;
   1:  PR[91,2] = PR[90,2] + -8.536;
   1:  PR[91,3] = PR[90,3] + 2.377;
   1:L PR[91] R[100]mm/sec CNT100;
   1:  PR[91,1] = PR[90,1] + -34.095;
   1:  PR[91,2] = PR[90,2] + -9.069;
   1:  PR[91,3] = PR[90,3] + 2.383;
   1:L PR[91] R[100]mm/sec CNT100;
   1:  PR[91,1] = PR[90,1] + -33.742;
   1:  PR[91,2] = PR[90,2] + -9.568;
   1:  PR[91,3] = PR[90,3] + 2.387;
   1:L PR[91] R[100]mm/sec CNT100;
   1:  PR[91,1] = PR[90,1] + -33.374;
   1:  PR[91,2] = PR[90,2] + -10.052;
   1:  PR[91,3] = PR[90,3] + 2.390;
   1:L PR[91] R[100]mm/sec CNT100;
   1:  PR[91,1] = PR[90,1] + -32.787;
   1:  PR[91,2] = PR[90,2] + -10.758;
   1:  PR[91,3] = PR[90,3] + 2.394;
   1:L PR[91] R[100]mm/sec CNT100;
   1:  PR[91,1] = PR[90,1] + -31.932;
   1:  PR[91,2] = PR[90,2] + -11.658;
   1:  PR[91,3] = PR[90,3] + 2.400;
   1:L PR[91] R[100]mm/sec CNT100;
   1:  PR[91,1] = PR[90,1] + -31.041;
   1:  PR[91,2] = PR[90,2] + -12.468;
   1:  PR[91,3] = PR[90,3] + 2.407;
   1:L PR[91] R[100]mm/sec CNT100;
   1:  PR[91,1] = PR[90,1] + -30.081;
   1:  PR[91,2] = PR[90,2] + -13.224;
   1:  PR[91,3] = PR[90,3] + 2.415;
   1:L PR[91] R[100]mm/sec CNT100;
   1:  PR[91,1] = PR[90,1] + -29.068;
   1:  PR[91,2] = PR[90,2] + -13.908;
   1:  PR[91,3] = PR[90,3] + 2.422;
   1:L PR[91] R[100]mm/sec CNT100;
   1:  PR[91,1] = PR[90,1] + -28.008;
   1:  PR[91,2] = PR[90,2] + -14.518;
   1:  PR[91,3] = PR[90,3] + 2.429;
   1:L PR[91] R[100]mm/sec CNT100;
   1:  PR[91,1] = PR[90,1] + -26.908;
   1:  PR[91,2] = PR[90,2] + -15.048;
   1:  PR[91,3] = PR[90,3] + 2.437;
   1:L PR[91] R[100]mm/sec CNT100;
   1:  PR[91,1] = PR[90,1] + -25.771;
   1:  PR[91,2] = PR[90,2] + -15.499;
   1:  PR[91,3] = PR[90,3] + 2.444;
   1:L PR[91] R[100]mm/sec CNT100;
   1:  PR[91,1] = PR[90,1] + -24.606;
   1:  PR[91,2] = PR[90,2] + -15.865;
   1:  PR[91,3] = PR[90,3] + 2.452;
   1:L PR[91] R[100]mm/sec CNT100;
   1:  PR[91,1] = PR[90,1] + -23.416;
   1:  PR[91,2] = PR[90,2] + -16.147;
   1:  PR[91,3] = PR[90,3] + 2.459;
   1:L PR[91] R[100]mm/sec CNT100;
   1:  PR[91,1] = PR[90,1] + -22.210;
   1:  PR[91,2] = PR[90,2] + -16.342;
   1:  PR[91,3] = PR[90,3] + 2.467;
   1:L PR[91] R[100]mm/sec CNT100;
   1:  PR[91,1] = PR[90,1] + -20.992;
   1:  PR[91,2] = PR[90,2] + -16.449;
   1:  PR[91,3] = PR[90,3] + 2.474;
   1:L PR[91] R[100]mm/sec CNT100;
   1:  PR[91,1] = PR[90,1] + -19.771;
   1:  PR[91,2] = PR[90,2] + -16.468;
   1:  PR[91,3] = PR[90,3] + 2.481;
   1:L PR[91] R[100]mm/sec CNT100;
   1:  PR[91,1] = PR[90,1] + -18.550;
   1:  PR[91,2] = PR[90,2] + -16.399;
   1:  PR[91,3] = PR[90,3] + 2.489;
   1:L PR[91] R[100]mm/sec CNT100;
   1:  PR[91,1] = PR[90,1] + -17.337;
   1:  PR[91,2] = PR[90,2] + -16.241;
   1:  PR[91,3] = PR[90,3] + 2.496;
   1:L PR[91] R[100]mm/sec CNT100;
   1:  PR[91,1] = PR[90,1] + -16.436;
   1:  PR[91,2] = PR[90,2] + -16.063;
   1:  PR[91,3] = PR[90,3] + 2.504;
   1:L PR[91] R[100]mm/sec CNT100;
   1:  PR[91,1] = PR[90,1] + -15.847;
   1:  PR[91,2] = PR[90,2] + -15.920;
   1:  PR[91,3] = PR[90,3] + 2.509;
   1:L PR[91] R[100]mm/sec CNT100;
   1:  PR[91,1] = PR[90,1] + -14.966;
   1:  PR[91,2] = PR[90,2] + -15.667;
   1:  PR[91,3] = PR[90,3] + 2.513;
   1:L PR[91] R[100]mm/sec CNT100;
   1:  PR[91,1] = PR[90,1] + -13.815;
   1:  PR[91,2] = PR[90,2] + -15.252;
   1:  PR[91,3] = PR[90,3] + 2.519;
   1:L PR[91] R[100]mm/sec CNT100;
   1:  PR[91,1] = PR[90,1] + -12.692;
   1:  PR[91,2] = PR[90,2] + -14.753;
   1:  PR[91,3] = PR[90,3] + 2.526;
   1:L PR[91] R[100]mm/sec CNT100;
   1:  PR[91,1] = PR[90,1] + -12.253;
   1:  PR[91,2] = PR[90,2] + -14.529;
   1:  PR[91,3] = PR[90,3] + 2.533;
   1:L PR[91] R[100]mm/sec CNT100;
   1:  PR[91,1] = PR[90,1] + -11.624;
   1:  PR[91,2] = PR[90,2] + -14.182;
   1:  PR[91,3] = PR[90,3] + 2.536;
   1:L PR[91] R[100]mm/sec CNT100;
   1:  PR[91,1] = PR[90,1] + -10.585;
   1:  PR[91,2] = PR[90,2] + -13.526;
   1:  PR[91,3] = PR[90,3] + 2.541;
   1:L PR[91] R[100]mm/sec CNT100;
   1:  PR[91,1] = PR[90,1] + -9.844;
   1:  PR[91,2] = PR[90,2] + -12.986;
   1:  PR[91,3] = PR[90,3] + 2.548;
   1:L PR[91] R[100]mm/sec CNT100;
   1:  PR[91,1] = PR[90,1] + -9.368;
   1:  PR[91,2] = PR[90,2] + -12.608;
   1:  PR[91,3] = PR[90,3] + 2.554;
   1:L PR[91] R[100]mm/sec CNT100;
   1:  PR[91,1] = PR[90,1] + -8.903;
   1:  PR[91,2] = PR[90,2] + -12.210;
   1:  PR[91,3] = PR[90,3] + 2.558;
   1:L PR[91] R[100]mm/sec CNT100;
   1:  PR[91,1] = PR[90,1] + -8.278;
   1:  PR[91,2] = PR[90,2] + -11.630;
   1:  PR[91,3] = PR[90,3] + 2.561;
   1:L PR[91] R[100]mm/sec CNT100;
   1:  PR[91,1] = PR[90,1] + -7.808;
   1:  PR[91,2] = PR[90,2] + -11.150;
   1:  PR[91,3] = PR[90,3] + 2.566;
   1:L PR[91] R[100]mm/sec CNT100;
   1:  PR[91,1] = PR[90,1] + -7.196;
   1:  PR[91,2] = PR[90,2] + -10.458;
   1:  PR[91,3] = PR[90,3] + 2.570;
   1:L PR[91] R[100]mm/sec CNT100;
   1:  PR[91,1] = PR[90,1] + -6.813;
   1:  PR[91,2] = PR[90,2] + -9.987;
   1:  PR[91,3] = PR[90,3] + 2.576;
   1:L PR[91] R[100]mm/sec CNT100;
   1:  PR[91,1] = PR[90,1] + -6.446;
   1:  PR[91,2] = PR[90,2] + -9.500;
   1:  PR[91,3] = PR[90,3] + 2.580;
   1:L PR[91] R[100]mm/sec CNT100;
   1:  PR[91,1] = PR[90,1] + -5.934;
   1:  PR[91,2] = PR[90,2] + -8.758;
   1:  PR[91,3] = PR[90,3] + 2.583;
   1:L PR[91] R[100]mm/sec CNT100;
   1:  PR[91,1] = PR[90,1] + -5.605;
   1:  PR[91,2] = PR[90,2] + -8.229;
   1:  PR[91,3] = PR[90,3] + 2.589;
   1:L PR[91] R[100]mm/sec CNT100;
   1:  PR[91,1] = PR[90,1] + -5.015;
   1:  PR[91,2] = PR[90,2] + -7.153;
   1:  PR[91,3] = PR[90,3] + 2.593;
   1:L PR[91] R[100]mm/sec CNT100;
   1:  PR[91,1] = PR[90,1] + -4.506;
   1:  PR[91,2] = PR[90,2] + -6.039;
   1:  PR[91,3] = PR[90,3] + 2.600;
   1:L PR[91] R[100]mm/sec CNT100;
   1:  PR[91,1] = PR[90,1] + -4.181;
   1:  PR[91,2] = PR[90,2] + -5.182;
   1:  PR[91,3] = PR[90,3] + 2.608;
   1:L PR[91] R[100]mm/sec CNT100;
   1:  PR[91,1] = PR[90,1] + -3.990;
   1:  PR[91,2] = PR[90,2] + -4.608;
   1:  PR[91,3] = PR[90,3] + 2.613;
   1:L PR[91] R[100]mm/sec CNT100;
   1:  PR[91,1] = PR[90,1] + -3.738;
   1:  PR[91,2] = PR[90,2] + -3.725;
   1:  PR[91,3] = PR[90,3] + 2.617;
   1:L PR[91] R[100]mm/sec CNT100;
   1:  PR[91,1] = PR[90,1] + -3.384;
   1:  PR[91,2] = PR[90,2] + -2.138;
   1:  PR[91,3] = PR[90,3] + 2.622;
   1:L PR[91] R[100]mm/sec CNT100;
   1:  PR[91,1] = PR[90,1] + -3.176;
   1:  PR[91,2] = PR[90,2] + -1.639;
   1:  PR[91,3] = PR[90,3] + 2.632;
   1:L PR[91] R[100]mm/sec CNT100;
   1:  PR[91,1] = PR[90,1] + -2.892;
   1:  PR[91,2] = PR[90,2] + -1.194;
   1:  PR[91,3] = PR[90,3] + 2.636;
   1:L PR[91] R[100]mm/sec CNT100;
   1:  PR[91,1] = PR[90,1] + -2.708;
   1:  PR[91,2] = PR[90,2] + -0.974;
   1:  PR[91,3] = PR[90,3] + 2.639;
   1:L PR[91] R[100]mm/sec CNT100;
   1:  PR[91,1] = PR[90,1] + -2.417;
   1:  PR[91,2] = PR[90,2] + -0.692;
   1:  PR[91,3] = PR[90,3] + 2.641;
   1:L PR[91] R[100]mm/sec CNT100;
   1:  PR[91,1] = PR[90,1] + -1.978;
   1:  PR[91,2] = PR[90,2] + -0.385;
   1:  PR[91,3] = PR[90,3] + 2.643;
   1:L PR[91] R[100]mm/sec CNT100;
   1:  PR[91,1] = PR[90,1] + -1.487;
   1:  PR[91,2] = PR[90,2] + -0.157;
   1:  PR[91,3] = PR[90,3] + 2.646;
   1:L PR[91] R[100]mm/sec CNT100;
   1:  PR[91,1] = PR[90,1] + -0.968;
   1:  PR[91,2] = PR[90,2] + -0.018;
   1:  PR[91,3] = PR[90,3] + 2.650;
   1:L PR[91] R[100]mm/sec CNT100;
   1:  PR[91,1] = PR[90,1] + -0.569;
   1:  PR[91,2] = PR[90,2] + 0.023;
   1:  PR[91,3] = PR[90,3] + 2.653;
   1:L PR[91] R[100]mm/sec CNT100;
   1:  PR[91,1] = PR[90,1] + 0.209;
   1:  PR[91,2] = PR[90,2] + 0.028;
   1:  PR[91,3] = PR[90,3] + 2.655;
   1:L PR[91] R[100]mm/sec CNT100;
   1:  PR[91] = PR[90];
   1:  PR[91,1] = PR[90,1] + 0.499;
   1:  PR[91,2] = PR[90,2] + 0.011;
   1:  PR[91,3] = PR[90,3] + 3.990;
   1:L PR[91] R[100]mm/sec CNT100;
   1:  PR[91,1] = PR[90,1] + 0.740;
   1:  PR[91,2] = PR[90,2] + -0.020;
   1:  PR[91,3] = PR[90,3] + 2.662;
   1:L PR[91] R[100]mm/sec CNT100;
   1:  PR[91,1] = PR[90,1] + 1.240;
   1:  PR[91,2] = PR[90,2] + -0.154;
   1:  PR[91,3] = PR[90,3] + 2.663;
   1:L PR[91] R[100]mm/sec CNT100;
   1:  PR[91,1] = PR[90,1] + 1.547;
   1:  PR[91,2] = PR[90,2] + -0.286;
   1:  PR[91,3] = PR[90,3] + 2.666;
   1:L PR[91] R[100]mm/sec CNT100;
   1:  PR[91,1] = PR[90,1] + 1.922;
   1:  PR[91,2] = PR[90,2] + -0.502;
   1:  PR[91,3] = PR[90,3] + 2.668;
   1:L PR[91] R[100]mm/sec CNT100;
   1:  PR[91,1] = PR[90,1] + 2.181;
   1:  PR[91,2] = PR[90,2] + -0.696;
   1:  PR[91,3] = PR[90,3] + 2.671;
   1:L PR[91] R[100]mm/sec CNT100;
   1:  PR[91,1] = PR[90,1] + 2.408;
   1:  PR[91,2] = PR[90,2] + -0.908;
   1:  PR[91,3] = PR[90,3] + 2.673;
   1:L PR[91] R[100]mm/sec CNT100;
   1:  PR[91,1] = PR[90,1] + 2.572;
   1:  PR[91,2] = PR[90,2] + -1.087;
   1:  PR[91,3] = PR[90,3] + 2.675;
   1:L PR[91] R[100]mm/sec CNT100;
   1:  PR[91,1] = PR[90,1] + 2.869;
   1:  PR[91,2] = PR[90,2] + -1.511;
   1:  PR[91,3] = PR[90,3] + 2.676;
   1:L PR[91] R[100]mm/sec CNT100;
   1:  PR[91,1] = PR[90,1] + 3.020;
   1:  PR[91,2] = PR[90,2] + -1.809;
   1:  PR[91,3] = PR[90,3] + 2.680;
   1:L PR[91] R[100]mm/sec CNT100;
   1:  PR[91,1] = PR[90,1] + 3.170;
   1:  PR[91,2] = PR[90,2] + -2.220;
   1:  PR[91,3] = PR[90,3] + 2.682;
   1:L PR[91] R[100]mm/sec CNT100;
   1:  PR[91,1] = PR[90,1] + 3.500;
   1:  PR[91,2] = PR[90,2] + -3.728;
   1:  PR[91,3] = PR[90,3] + 2.684;
   1:L PR[91] R[100]mm/sec CNT100;
   1:  PR[91,1] = PR[90,1] + 3.691;
   1:  PR[91,2] = PR[90,2] + -4.414;
   1:  PR[91,3] = PR[90,3] + 2.694;
   1:L PR[91] R[100]mm/sec CNT100;
   1:  PR[91,1] = PR[90,1] + 3.841;
   1:  PR[91,2] = PR[90,2] + -4.896;
   1:  PR[91,3] = PR[90,3] + 2.698;
   1:L PR[91] R[100]mm/sec CNT100;
   1:  PR[91,1] = PR[90,1] + 4.071;
   1:  PR[91,2] = PR[90,2] + -5.542;
   1:  PR[91,3] = PR[90,3] + 2.701;
   1:L PR[91] R[100]mm/sec CNT100;
   1:  PR[91,1] = PR[90,1] + 4.266;
   1:  PR[91,2] = PR[90,2] + -6.037;
   1:  PR[91,3] = PR[90,3] + 2.705;
   1:L PR[91] R[100]mm/sec CNT100;
   1:  PR[91,1] = PR[90,1] + 4.779;
   1:  PR[91,2] = PR[90,2] + -7.157;
   1:  PR[91,3] = PR[90,3] + 2.708;
   1:L PR[91] R[100]mm/sec CNT100;
   1:  PR[91,1] = PR[90,1] + 5.113;
   1:  PR[91,2] = PR[90,2] + -7.786;
   1:  PR[91,3] = PR[90,3] + 2.716;
   1:L PR[91] R[100]mm/sec CNT100;
   1:  PR[91,1] = PR[90,1] + 5.364;
   1:  PR[91,2] = PR[90,2] + -8.225;
   1:  PR[91,3] = PR[90,3] + 2.720;
   1:L PR[91] R[100]mm/sec CNT100;
   1:  PR[91,1] = PR[90,1] + 5.690;
   1:  PR[91,2] = PR[90,2] + -8.751;
   1:  PR[91,3] = PR[90,3] + 2.723;
   1:L PR[91] R[100]mm/sec CNT100;
   1:  PR[91,1] = PR[90,1] + 6.025;
   1:  PR[91,2] = PR[90,2] + -9.248;
   1:  PR[91,3] = PR[90,3] + 2.727;
   1:L PR[91] R[100]mm/sec CNT100;
   1:  PR[91,1] = PR[90,1] + 6.764;
   1:  PR[91,2] = PR[90,2] + -10.228;
   1:  PR[91,3] = PR[90,3] + 2.731;
   1:L PR[91] R[100]mm/sec CNT100;
   1:  PR[91,1] = PR[90,1] + 7.572;
   1:  PR[91,2] = PR[90,2] + -11.152;
   1:  PR[91,3] = PR[90,3] + 2.738;
   1:L PR[91] R[100]mm/sec CNT100;
   1:  PR[91,1] = PR[90,1] + 8.011;
   1:  PR[91,2] = PR[90,2] + -11.602;
   1:  PR[91,3] = PR[90,3] + 2.746;
   1:L PR[91] R[100]mm/sec CNT100;
   1:  PR[91,1] = PR[90,1] + 8.432;
   1:  PR[91,2] = PR[90,2] + -12.004;
   1:  PR[91,3] = PR[90,3] + 2.749;
   1:L PR[91] R[100]mm/sec CNT100;
   1:  PR[91,1] = PR[90,1] + 9.365;
   1:  PR[91,2] = PR[90,2] + -12.802;
   1:  PR[91,3] = PR[90,3] + 2.753;
   1:L PR[91] R[100]mm/sec CNT100;
   1:  PR[91,1] = PR[90,1] + 10.349;
   1:  PR[91,2] = PR[90,2] + -13.527;
   1:  PR[91,3] = PR[90,3] + 2.760;
   1:L PR[91] R[100]mm/sec CNT100;
   1:  PR[91,1] = PR[90,1] + 11.387;
   1:  PR[91,2] = PR[90,2] + -14.182;
   1:  PR[91,3] = PR[90,3] + 2.768;
   1:L PR[91] R[100]mm/sec CNT100;
   1:  PR[91,1] = PR[90,1] + 11.949;
   1:  PR[91,2] = PR[90,2] + -14.495;
   1:  PR[91,3] = PR[90,3] + 2.775;
   1:L PR[91] R[100]mm/sec CNT100;
   1:  PR[91,1] = PR[90,1] + 12.455;
   1:  PR[91,2] = PR[90,2] + -14.754;
   1:  PR[91,3] = PR[90,3] + 2.779;
   1:L PR[91] R[100]mm/sec CNT100;
   1:  PR[91,1] = PR[90,1] + 13.577;
   1:  PR[91,2] = PR[90,2] + -15.252;
   1:  PR[91,3] = PR[90,3] + 2.783;
   1:L PR[91] R[100]mm/sec CNT100;
   1:  PR[91,1] = PR[90,1] + 14.727;
   1:  PR[91,2] = PR[90,2] + -15.667;
   1:  PR[91,3] = PR[90,3] + 2.790;
   1:L PR[91] R[100]mm/sec CNT100;
   1:  PR[91,1] = PR[90,1] + 15.907;
   1:  PR[91,2] = PR[90,2] + -15.998;
   1:  PR[91,3] = PR[90,3] + 2.798;
   1:L PR[91] R[100]mm/sec CNT100;
   1:  PR[91,1] = PR[90,1] + 16.603;
   1:  PR[91,2] = PR[90,2] + -16.150;
   1:  PR[91,3] = PR[90,3] + 2.805;
   1:L PR[91] R[100]mm/sec CNT100;
   1:  PR[91,1] = PR[90,1] + 17.095;
   1:  PR[91,2] = PR[90,2] + -16.241;
   1:  PR[91,3] = PR[90,3] + 2.809;
   1:L PR[91] R[100]mm/sec CNT100;
   1:  PR[91,1] = PR[90,1] + 18.313;
   1:  PR[91,2] = PR[90,2] + -16.399;
   1:  PR[91,3] = PR[90,3] + 2.812;
   1:L PR[91] R[100]mm/sec CNT100;
   1:  PR[91,1] = PR[90,1] + 19.533;
   1:  PR[91,2] = PR[90,2] + -16.468;
   1:  PR[91,3] = PR[90,3] + 2.820;
   1:L PR[91] R[100]mm/sec CNT100;
   1:  PR[91,1] = PR[90,1] + 20.759;
   1:  PR[91,2] = PR[90,2] + -16.449;
   1:  PR[91,3] = PR[90,3] + 2.827;
   1:L PR[91] R[100]mm/sec CNT100;
   1:  PR[91,1] = PR[90,1] + 21.469;
   1:  PR[91,2] = PR[90,2] + -16.396;
   1:  PR[91,3] = PR[90,3] + 2.835;
   1:L PR[91] R[100]mm/sec CNT100;
   1:  PR[91,1] = PR[90,1] + 21.967;
   1:  PR[91,2] = PR[90,2] + -16.343;
   1:  PR[91,3] = PR[90,3] + 2.839;
   1:L PR[91] R[100]mm/sec CNT100;
   1:  PR[91,1] = PR[90,1] + 23.179;
   1:  PR[91,2] = PR[90,2] + -16.147;
   1:  PR[91,3] = PR[90,3] + 2.842;
   1:L PR[91] R[100]mm/sec CNT100;
   1:  PR[91,1] = PR[90,1] + 24.372;
   1:  PR[91,2] = PR[90,2] + -15.864;
   1:  PR[91,3] = PR[90,3] + 2.849;
   1:L PR[91] R[100]mm/sec CNT100;
   1:  PR[91,1] = PR[90,1] + 25.054;
   1:  PR[91,2] = PR[90,2] + -15.659;
   1:  PR[91,3] = PR[90,3] + 2.857;
   1:L PR[91] R[100]mm/sec CNT100;
   1:  PR[91,1] = PR[90,1] + 25.529;
   1:  PR[91,2] = PR[90,2] + -15.500;
   1:  PR[91,3] = PR[90,3] + 2.861;
   1:L PR[91] R[100]mm/sec CNT100;
   1:  PR[91,1] = PR[90,1] + 26.670;
   1:  PR[91,2] = PR[90,2] + -15.048;
   1:  PR[91,3] = PR[90,3] + 2.864;
   1:L PR[91] R[100]mm/sec CNT100;
   1:  PR[91,1] = PR[90,1] + 27.771;
   1:  PR[91,2] = PR[90,2] + -14.517;
   1:  PR[91,3] = PR[90,3] + 2.872;
   1:L PR[91] R[100]mm/sec CNT100;
   1:  PR[91,1] = PR[90,1] + 28.834;
   1:  PR[91,2] = PR[90,2] + -13.906;
   1:  PR[91,3] = PR[90,3] + 2.879;
   1:L PR[91] R[100]mm/sec CNT100;
   1:  PR[91,1] = PR[90,1] + 29.429;
   1:  PR[91,2] = PR[90,2] + -13.515;
   1:  PR[91,3] = PR[90,3] + 2.887;
   1:L PR[91] R[100]mm/sec CNT100;
   1:  PR[91,1] = PR[90,1] + 29.839;
   1:  PR[91,2] = PR[90,2] + -13.227;
   1:  PR[91,3] = PR[90,3] + 2.891;
   1:L PR[91] R[100]mm/sec CNT100;
   1:  PR[91,1] = PR[90,1] + 30.803;
   1:  PR[91,2] = PR[90,2] + -12.468;
   1:  PR[91,3] = PR[90,3] + 2.894;
   1:L PR[91] R[100]mm/sec CNT100;
   1:  PR[91,1] = PR[90,1] + 31.707;
   1:  PR[91,2] = PR[90,2] + -11.645;
   1:  PR[91,3] = PR[90,3] + 2.901;
   1:L PR[91] R[100]mm/sec CNT100;
   1:  PR[91,1] = PR[90,1] + 32.551;
   1:  PR[91,2] = PR[90,2] + -10.756;
   1:  PR[91,3] = PR[90,3] + 2.909;
   1:L PR[91] R[100]mm/sec CNT100;
   1:  PR[91,1] = PR[90,1] + 33.010;
   1:  PR[91,2] = PR[90,2] + -10.210;
   1:  PR[91,3] = PR[90,3] + 2.916;
   1:L PR[91] R[100]mm/sec CNT100;
   1:  PR[91,1] = PR[90,1] + 33.321;
   1:  PR[91,2] = PR[90,2] + -9.818;
   1:  PR[91,3] = PR[90,3] + 2.921;
   1:L PR[91] R[100]mm/sec CNT100;
   1:  PR[91,1] = PR[90,1] + 34.034;
   1:  PR[91,2] = PR[90,2] + -8.807;
   1:  PR[91,3] = PR[90,3] + 2.924;
   1:L PR[91] R[100]mm/sec CNT100;
   1:  PR[91,1] = PR[90,1] + 34.660;
   1:  PR[91,2] = PR[90,2] + -7.769;
   1:  PR[91,3] = PR[90,3] + 2.931;
   1:L PR[91] R[100]mm/sec CNT100;
   1:  PR[91,1] = PR[90,1] + 35.216;
   1:  PR[91,2] = PR[90,2] + -6.675;
   1:  PR[91,3] = PR[90,3] + 2.939;
   1:L PR[91] R[100]mm/sec CNT100;
   1:  PR[91,1] = PR[90,1] + 35.478;
   1:  PR[91,2] = PR[90,2] + -6.077;
   1:  PR[91,3] = PR[90,3] + 2.946;
   1:L PR[91] R[100]mm/sec CNT100;
   1:  PR[91,1] = PR[90,1] + 35.685;
   1:  PR[91,2] = PR[90,2] + -5.558;
   1:  PR[91,3] = PR[90,3] + 2.950;
   1:L PR[91] R[100]mm/sec CNT100;
   1:  PR[91,1] = PR[90,1] + 36.079;
   1:  PR[91,2] = PR[90,2] + -4.391;
   1:  PR[91,3] = PR[90,3] + 2.953;
   1:L PR[91] R[100]mm/sec CNT100;
   1:  PR[91,1] = PR[90,1] + 36.265;
   1:  PR[91,2] = PR[90,2] + -3.709;
   1:  PR[91,3] = PR[90,3] + 2.961;
   1:L PR[91] R[100]mm/sec CNT100;
   1:  PR[91,1] = PR[90,1] + 36.494;
   1:  PR[91,2] = PR[90,2] + -2.668;
   1:  PR[91,3] = PR[90,3] + 2.965;
   1:L PR[91] R[100]mm/sec CNT100;
   1:  PR[91,1] = PR[90,1] + 36.604;
   1:  PR[91,2] = PR[90,2] + -2.010;
   1:  PR[91,3] = PR[90,3] + 2.972;
   1:L PR[91] R[100]mm/sec CNT100;
   1:  PR[91,1] = PR[90,1] + 36.691;
   1:  PR[91,2] = PR[90,2] + -1.298;
   1:  PR[91,3] = PR[90,3] + 2.976;
   1:L PR[91] R[100]mm/sec CNT100;
   1:  PR[91,1] = PR[90,1] + 36.736;
   1:  PR[91,2] = PR[90,2] + -0.795;
   1:  PR[91,3] = PR[90,3] + 2.980;
   1:L PR[91] R[100]mm/sec CNT100;
   1:  PR[91,1] = PR[90,1] + 36.770;
   1:  PR[91,2] = PR[90,2] + -0.164;
   1:  PR[91,3] = PR[90,3] + 2.983;
   1:L PR[91] R[100]mm/sec CNT100;
   1:  PR[91,1] = PR[90,1] + 36.781;
   1:  PR[91,2] = PR[90,2] + 0.426;
   1:  PR[91,3] = PR[90,3] + 2.987;
   1:L PR[91] R[100]mm/sec CNT100;
   1:  PR[91,1] = PR[90,1] + 36.764;
   1:  PR[91,2] = PR[90,2] + 1.139;
   1:  PR[91,3] = PR[90,3] + 2.991;
   1:L PR[91] R[100]mm/sec CNT100;
   1:  PR[91,1] = PR[90,1] + 36.690;
   1:  PR[91,2] = PR[90,2] + 2.159;
   1:  PR[91,3] = PR[90,3] + 2.995;
   1:L PR[91] R[100]mm/sec CNT100;
   1:  PR[91,1] = PR[90,1] + 36.604;
   1:  PR[91,2] = PR[90,2] + 2.864;
   1:  PR[91,3] = PR[90,3] + 3.001;
   1:L PR[91] R[100]mm/sec CNT100;
   1:  PR[91,1] = PR[90,1] + 36.485;
   1:  PR[91,2] = PR[90,2] + 3.565;
   1:  PR[91,3] = PR[90,3] + 3.005;
   1:L PR[91] R[100]mm/sec CNT100;
   1:  PR[91,1] = PR[90,1] + 36.265;
   1:  PR[91,2] = PR[90,2] + 4.564;
   1:  PR[91,3] = PR[90,3] + 3.010;
   1:L PR[91] R[100]mm/sec CNT100;
   1:  PR[91,1] = PR[90,1] + 36.078;
   1:  PR[91,2] = PR[90,2] + 5.251;
   1:  PR[91,3] = PR[90,3] + 3.016;
   1:L PR[91] R[100]mm/sec CNT100;
   1:  PR[91,1] = PR[90,1] + 35.899;
   1:  PR[91,2] = PR[90,2] + 5.815;
   1:  PR[91,3] = PR[90,3] + 3.020;
   1:L PR[91] R[100]mm/sec CNT100;
   1:  PR[91,1] = PR[90,1] + 35.688;
   1:  PR[91,2] = PR[90,2] + 6.406;
   1:  PR[91,3] = PR[90,3] + 3.024;
   1:L PR[91] R[100]mm/sec CNT100;
   1:  PR[91,1] = PR[90,1] + 35.420;
   1:  PR[91,2] = PR[90,2] + 7.067;
   1:  PR[91,3] = PR[90,3] + 3.028;
   1:L PR[91] R[100]mm/sec CNT100;
   1:  PR[91,1] = PR[90,1] + 34.990;
   1:  PR[91,2] = PR[90,2] + 7.994;
   1:  PR[91,3] = PR[90,3] + 3.032;
   1:L PR[91] R[100]mm/sec CNT100;
   1:  PR[91,1] = PR[90,1] + 34.659;
   1:  PR[91,2] = PR[90,2] + 8.625;
   1:  PR[91,3] = PR[90,3] + 3.038;
   1:L PR[91] R[100]mm/sec CNT100;
   1:  PR[91,1] = PR[90,1] + 34.301;
   1:  PR[91,2] = PR[90,2] + 9.238;
   1:  PR[91,3] = PR[90,3] + 3.043;
   1:L PR[91] R[100]mm/sec CNT100;
   1:  PR[91,1] = PR[90,1] + 33.741;
   1:  PR[91,2] = PR[90,2] + 10.094;
   1:  PR[91,3] = PR[90,3] + 3.047;
   1:L PR[91] R[100]mm/sec CNT100;
   1:  PR[91,1] = PR[90,1] + 33.324;
   1:  PR[91,2] = PR[90,2] + 10.669;
   1:  PR[91,3] = PR[90,3] + 3.053;
   1:L PR[91] R[100]mm/sec CNT100;
   1:  PR[91,1] = PR[90,1] + 32.889;
   1:  PR[91,2] = PR[90,2] + 11.214;
   1:  PR[91,3] = PR[90,3] + 3.057;
   1:L PR[91] R[100]mm/sec CNT100;
   1:  PR[91,1] = PR[90,1] + 32.550;
   1:  PR[91,2] = PR[90,2] + 11.613;
   1:  PR[91,3] = PR[90,3] + 3.062;
   1:L PR[91] R[100]mm/sec CNT100;
   1:  PR[91,1] = PR[90,1] + 32.066;
   1:  PR[91,2] = PR[90,2] + 12.135;
   1:  PR[91,3] = PR[90,3] + 3.065;
   1:L PR[91] R[100]mm/sec CNT100;
   1:  PR[91,1] = PR[90,1] + 31.335;
   1:  PR[91,2] = PR[90,2] + 12.851;
   1:  PR[91,3] = PR[90,3] + 3.069;
   1:L PR[91] R[100]mm/sec CNT100;
   1:  PR[91,1] = PR[90,1] + 30.803;
   1:  PR[91,2] = PR[90,2] + 13.323;
   1:  PR[91,3] = PR[90,3] + 3.075;
   1:L PR[91] R[100]mm/sec CNT100;
   1:  PR[91,1] = PR[90,1] + 30.246;
   1:  PR[91,2] = PR[90,2] + 13.773;
   1:  PR[91,3] = PR[90,3] + 3.080;
   1:L PR[91] R[100]mm/sec CNT100;
   1:  PR[91,1] = PR[90,1] + 29.843;
   1:  PR[91,2] = PR[90,2] + 14.079;
   1:  PR[91,3] = PR[90,3] + 3.084;
   1:L PR[91] R[100]mm/sec CNT100;
   1:  PR[91,1] = PR[90,1] + 29.341;
   1:  PR[91,2] = PR[90,2] + 14.432;
   1:  PR[91,3] = PR[90,3] + 3.087;
   1:L PR[91] R[100]mm/sec CNT100;
   1:  PR[91,1] = PR[90,1] + 28.835;
   1:  PR[91,2] = PR[90,2] + 14.760;
   1:  PR[91,3] = PR[90,3] + 3.091;
   1:L PR[91] R[100]mm/sec CNT100;
   1:  PR[91,1] = PR[90,1] + 27.767;
   1:  PR[91,2] = PR[90,2] + 15.374;
   1:  PR[91,3] = PR[90,3] + 3.094;
   1:L PR[91] R[100]mm/sec CNT100;
   1:  PR[91,1] = PR[90,1] + 27.135;
   1:  PR[91,2] = PR[90,2] + 15.690;
   1:  PR[91,3] = PR[90,3] + 3.102;
   1:L PR[91] R[100]mm/sec CNT100;
   1:  PR[91,1] = PR[90,1] + 26.198;
   1:  PR[91,2] = PR[90,2] + 16.100;
   1:  PR[91,3] = PR[90,3] + 3.106;
   1:L PR[91] R[100]mm/sec CNT100;
   1:  PR[91,1] = PR[90,1] + 25.534;
   1:  PR[91,2] = PR[90,2] + 16.354;
   1:  PR[91,3] = PR[90,3] + 3.112;
   1:L PR[91] R[100]mm/sec CNT100;
   1:  PR[91,1] = PR[90,1] + 24.859;
   1:  PR[91,2] = PR[90,2] + 16.576;
   1:  PR[91,3] = PR[90,3] + 3.117;
   1:L PR[91] R[100]mm/sec CNT100;
   1:  PR[91,1] = PR[90,1] + 23.873;
   1:  PR[91,2] = PR[90,2] + 16.847;
   1:  PR[91,3] = PR[90,3] + 3.121;
   1:L PR[91] R[100]mm/sec CNT100;
   1:  PR[91,1] = PR[90,1] + 23.182;
   1:  PR[91,2] = PR[90,2] + 17.002;
   1:  PR[91,3] = PR[90,3] + 3.127;
   1:L PR[91] R[100]mm/sec CNT100;
   1:  PR[91,1] = PR[90,1] + 21.969;
   1:  PR[91,2] = PR[90,2] + 17.198;
   1:  PR[91,3] = PR[90,3] + 3.132;
   1:L PR[91] R[100]mm/sec CNT100;
   1:  PR[91,1] = PR[90,1] + 21.265;
   1:  PR[91,2] = PR[90,2] + 17.269;
   1:  PR[91,3] = PR[90,3] + 3.139;
   1:L PR[91] R[100]mm/sec CNT100;
   1:  PR[91,1] = PR[90,1] + 20.244;
   1:  PR[91,2] = PR[90,2] + 17.322;
   1:  PR[91,3] = PR[90,3] + 3.143;
   1:L PR[91] R[100]mm/sec CNT100;
   1:  PR[91,1] = PR[90,1] + 19.533;
   1:  PR[91,2] = PR[90,2] + 17.324;
   1:  PR[91,3] = PR[90,3] + 3.150;
   1:L PR[91] R[100]mm/sec CNT100;
   1:  PR[91,1] = PR[90,1] + 18.823;
   1:  PR[91,2] = PR[90,2] + 17.293;
   1:  PR[91,3] = PR[90,3] + 3.154;
   1:L PR[91] R[100]mm/sec CNT100;
   1:  PR[91,1] = PR[90,1] + 17.805;
   1:  PR[91,2] = PR[90,2] + 17.198;
   1:  PR[91,3] = PR[90,3] + 3.158;
   1:L PR[91] R[100]mm/sec CNT100;
   1:  PR[91,1] = PR[90,1] + 17.105;
   1:  PR[91,2] = PR[90,2] + 17.098;
   1:  PR[91,3] = PR[90,3] + 3.164;
   1:L PR[91] R[100]mm/sec CNT100;
   1:  PR[91,1] = PR[90,1] + 15.903;
   1:  PR[91,2] = PR[90,2] + 16.852;
   1:  PR[91,3] = PR[90,3] + 3.169;
   1:L PR[91] R[100]mm/sec CNT100;
   1:  PR[91,1] = PR[90,1] + 14.727;
   1:  PR[91,2] = PR[90,2] + 16.522;
   1:  PR[91,3] = PR[90,3] + 3.176;
   1:L PR[91] R[100]mm/sec CNT100;
   1:  PR[91,1] = PR[90,1] + 13.577;
   1:  PR[91,2] = PR[90,2] + 16.107;
   1:  PR[91,3] = PR[90,3] + 3.184;
   1:L PR[91] R[100]mm/sec CNT100;
   1:  PR[91,1] = PR[90,1] + 12.460;
   1:  PR[91,2] = PR[90,2] + 15.611;
   1:  PR[91,3] = PR[90,3] + 3.191;
   1:L PR[91] R[100]mm/sec CNT100;
   1:  PR[91,1] = PR[90,1] + 11.379;
   1:  PR[91,2] = PR[90,2] + 15.033;
   1:  PR[91,3] = PR[90,3] + 3.198;
   1:L PR[91] R[100]mm/sec CNT100;
   1:  PR[91,1] = PR[90,1] + 10.785;
   1:  PR[91,2] = PR[90,2] + 14.670;
   1:  PR[91,3] = PR[90,3] + 3.206;
   1:L PR[91] R[100]mm/sec CNT100;
   1:  PR[91,1] = PR[90,1] + 10.350;
   1:  PR[91,2] = PR[90,2] + 14.384;
   1:  PR[91,3] = PR[90,3] + 3.210;
   1:L PR[91] R[100]mm/sec CNT100;
   1:  PR[91,1] = PR[90,1] + 9.771;
   1:  PR[91,2] = PR[90,2] + 13.968;
   1:  PR[91,3] = PR[90,3] + 3.213;
   1:L PR[91] R[100]mm/sec CNT100;
   1:  PR[91,1] = PR[90,1] + 8.971;
   1:  PR[91,2] = PR[90,2] + 13.332;
   1:  PR[91,3] = PR[90,3] + 3.218;
   1:L PR[91] R[100]mm/sec CNT100;
   1:  PR[91,1] = PR[90,1] + 8.436;
   1:  PR[91,2] = PR[90,2] + 12.863;
   1:  PR[91,3] = PR[90,3] + 3.224;
   1:L PR[91] R[100]mm/sec CNT100;
   1:  PR[91,1] = PR[90,1] + 7.921;
   1:  PR[91,2] = PR[90,2] + 12.366;
   1:  PR[91,3] = PR[90,3] + 3.228;
   1:L PR[91] R[100]mm/sec CNT100;
   1:  PR[91,1] = PR[90,1] + 7.568;
   1:  PR[91,2] = PR[90,2] + 12.003;
   1:  PR[91,3] = PR[90,3] + 3.232;
   1:L PR[91] R[100]mm/sec CNT100;
   1:  PR[91,1] = PR[90,1] + 7.156;
   1:  PR[91,2] = PR[90,2] + 11.549;
   1:  PR[91,3] = PR[90,3] + 3.236;
   1:L PR[91] R[100]mm/sec CNT100;
   1:  PR[91,1] = PR[90,1] + 6.767;
   1:  PR[91,2] = PR[90,2] + 11.087;
   1:  PR[91,3] = PR[90,3] + 3.239;
   1:L PR[91] R[100]mm/sec CNT100;
   1:  PR[91,1] = PR[90,1] + 6.026;
   1:  PR[91,2] = PR[90,2] + 10.104;
   1:  PR[91,3] = PR[90,3] + 3.243;
   1:L PR[91] R[100]mm/sec CNT100;
   1:  PR[91,1] = PR[90,1] + 5.631;
   1:  PR[91,2] = PR[90,2] + 9.510;
   1:  PR[91,3] = PR[90,3] + 3.250;
   1:L PR[91] R[100]mm/sec CNT100;
   1:  PR[91,1] = PR[90,1] + 5.364;
   1:  PR[91,2] = PR[90,2] + 9.080;
   1:  PR[91,3] = PR[90,3] + 3.255;
   1:L PR[91] R[100]mm/sec CNT100;
   1:  PR[91,1] = PR[90,1] + 5.069;
   1:  PR[91,2] = PR[90,2] + 8.565;
   1:  PR[91,3] = PR[90,3] + 3.258;
   1:L PR[91] R[100]mm/sec CNT100;
   1:  PR[91,1] = PR[90,1] + 4.778;
   1:  PR[91,2] = PR[90,2] + 8.010;
   1:  PR[91,3] = PR[90,3] + 3.261;
   1:L PR[91] R[100]mm/sec CNT100;
   1:  PR[91,1] = PR[90,1] + 4.471;
   1:  PR[91,2] = PR[90,2] + 7.361;
   1:  PR[91,3] = PR[90,3] + 3.265;
   1:L PR[91] R[100]mm/sec CNT100;
   1:  PR[91,1] = PR[90,1] + 4.269;
   1:  PR[91,2] = PR[90,2] + 6.899;
   1:  PR[91,3] = PR[90,3] + 3.270;
   1:L PR[91] R[100]mm/sec CNT100;
   1:  PR[91,1] = PR[90,1] + 4.012;
   1:  PR[91,2] = PR[90,2] + 6.235;
   1:  PR[91,3] = PR[90,3] + 3.273;
   1:L PR[91] R[100]mm/sec CNT100;
   1:  PR[91,1] = PR[90,1] + 3.688;
   1:  PR[91,2] = PR[90,2] + 5.261;
   1:  PR[91,3] = PR[90,3] + 3.277;
   1:L PR[91] R[100]mm/sec CNT100;
   1:  PR[91,1] = PR[90,1] + 3.500;
   1:  PR[91,2] = PR[90,2] + 4.583;
   1:  PR[91,3] = PR[90,3] + 3.283;
   1:L PR[91] R[100]mm/sec CNT100;
   1:  PR[91,1] = PR[90,1] + 3.170;
   1:  PR[91,2] = PR[90,2] + 3.074;
   1:  PR[91,3] = PR[90,3] + 3.287;
   1:L PR[91] R[100]mm/sec CNT100;
   1:  PR[91,1] = PR[90,1] + 3.007;
   1:  PR[91,2] = PR[90,2] + 2.633;
   1:  PR[91,3] = PR[90,3] + 3.297;
   1:L PR[91] R[100]mm/sec CNT100;
   1:  PR[91,1] = PR[90,1] + 2.872;
   1:  PR[91,2] = PR[90,2] + 2.372;
   1:  PR[91,3] = PR[90,3] + 3.300;
   1:L PR[91] R[100]mm/sec CNT100;
   1:  PR[91,1] = PR[90,1] + 2.696;
   1:  PR[91,2] = PR[90,2] + 2.104;
   1:  PR[91,3] = PR[90,3] + 3.301;
   1:L PR[91] R[100]mm/sec CNT100;
   1:  PR[91,1] = PR[90,1] + 2.417;
   1:  PR[91,2] = PR[90,2] + 1.772;
   1:  PR[91,3] = PR[90,3] + 3.303;
   1:L PR[91] R[100]mm/sec CNT100;
   1:  PR[91,1] = PR[90,1] + 2.174;
   1:  PR[91,2] = PR[90,2] + 1.544;
   1:  PR[91,3] = PR[90,3] + 3.306;
   1:L PR[91] R[100]mm/sec CNT100;
   1:  PR[91,1] = PR[90,1] + 1.739;
   1:  PR[91,2] = PR[90,2] + 1.240;
   1:  PR[91,3] = PR[90,3] + 3.308;
   1:L PR[91] R[100]mm/sec CNT100;
   1:  PR[91,1] = PR[90,1] + 1.249;
   1:  PR[91,2] = PR[90,2] + 1.012;
   1:  PR[91,3] = PR[90,3] + 3.311;
   1:L PR[91] R[100]mm/sec CNT100;
   1:  PR[91,1] = PR[90,1] + 0.736;
   1:  PR[91,2] = PR[90,2] + 0.875;
   1:  PR[91,3] = PR[90,3] + 3.315;
   1:L PR[91] R[100]mm/sec CNT100;
   1:  PR[91,1] = PR[90,1] + 0.409;
   1:  PR[91,2] = PR[90,2] + 0.836;
   1:  PR[91,3] = PR[90,3] + 3.318;
   1:L PR[91] R[100]mm/sec CNT100;
   1:  PR[91,1] = PR[90,1] + -0.451;
   1:  PR[91,2] = PR[90,2] + 0.827;
   1:  PR[91,3] = PR[90,3] + 3.320;
   1:L PR[91] R[100]mm/sec CNT100;
   1:  PR[91,1] = PR[90,1] + -0.965;
   1:  PR[91,2] = PR[90,2] + 0.872;
   1:  PR[91,3] = PR[90,3] + 3.325;
   1:L PR[91] R[100]mm/sec CNT100;
   1:  PR[91,1] = PR[90,1] + -1.478;
   1:  PR[91,2] = PR[90,2] + 1.010;
   1:  PR[91,3] = PR[90,3] + 3.328;
   1:L PR[91] R[100]mm/sec CNT100;
   1:  PR[91,1] = PR[90,1] + -1.785;
   1:  PR[91,2] = PR[90,2] + 1.141;
   1:  PR[91,3] = PR[90,3] + 3.331;
   1:L PR[91] R[100]mm/sec CNT100;
   1:  PR[91,1] = PR[90,1] + -2.160;
   1:  PR[91,2] = PR[90,2] + 1.357;
   1:  PR[91,3] = PR[90,3] + 3.333;
   1:L PR[91] R[100]mm/sec CNT100;
   1:  PR[91,1] = PR[90,1] + -2.420;
   1:  PR[91,2] = PR[90,2] + 1.551;
   1:  PR[91,3] = PR[90,3] + 3.336;
   1:L PR[91] R[100]mm/sec CNT100;
   1:  PR[91,1] = PR[90,1] + -2.646;
   1:  PR[91,2] = PR[90,2] + 1.763;
   1:  PR[91,3] = PR[90,3] + 3.338;
   1:L PR[91] R[100]mm/sec CNT100;
   1:  PR[91,1] = PR[90,1] + -2.810;
   1:  PR[91,2] = PR[90,2] + 1.942;
   1:  PR[91,3] = PR[90,3] + 3.340;
   1:L PR[91] R[100]mm/sec CNT100;
   1:  PR[91,1] = PR[90,1] + -3.106;
   1:  PR[91,2] = PR[90,2] + 2.364;
   1:  PR[91,3] = PR[90,3] + 3.341;
   1:L PR[91] R[100]mm/sec CNT100;
   1:  PR[91,1] = PR[90,1] + -3.246;
   1:  PR[91,2] = PR[90,2] + 2.633;
   1:  PR[91,3] = PR[90,3] + 3.345;
   1:L PR[91] R[100]mm/sec CNT100;
   1:  PR[91,1] = PR[90,1] + -3.408;
   1:  PR[91,2] = PR[90,2] + 3.074;
   1:  PR[91,3] = PR[90,3] + 3.346;
   1:L PR[91] R[100]mm/sec CNT100;
   1:  PR[91,1] = PR[90,1] + -3.738;
   1:  PR[91,2] = PR[90,2] + 4.583;
   1:  PR[91,3] = PR[90,3] + 3.349;
   1:L PR[91] R[100]mm/sec CNT100;
   1:  PR[91,1] = PR[90,1] + -3.929;
   1:  PR[91,2] = PR[90,2] + 5.269;
   1:  PR[91,3] = PR[90,3] + 3.359;
   1:L PR[91] R[100]mm/sec CNT100;
   1:  PR[91,1] = PR[90,1] + -4.079;
   1:  PR[91,2] = PR[90,2] + 5.747;
   1:  PR[91,3] = PR[90,3] + 3.363;
   1:L PR[91] R[100]mm/sec CNT100;
   1:  PR[91,1] = PR[90,1] + -4.507;
   1:  PR[91,2] = PR[90,2] + 6.897;
   1:  PR[91,3] = PR[90,3] + 3.366;
   1:L PR[91] R[100]mm/sec CNT100;
   1:  PR[91,1] = PR[90,1] + -5.018;
   1:  PR[91,2] = PR[90,2] + 8.014;
   1:  PR[91,3] = PR[90,3] + 3.373;
   1:L PR[91] R[100]mm/sec CNT100;
   1:  PR[91,1] = PR[90,1] + -5.308;
   1:  PR[91,2] = PR[90,2] + 8.565;
   1:  PR[91,3] = PR[90,3] + 3.381;
   1:L PR[91] R[100]mm/sec CNT100;
   1:  PR[91,1] = PR[90,1] + -5.600;
   1:  PR[91,2] = PR[90,2] + 9.076;
   1:  PR[91,3] = PR[90,3] + 3.385;
   1:L PR[91] R[100]mm/sec CNT100;
   1:  PR[91,1] = PR[90,1] + -6.266;
   1:  PR[91,2] = PR[90,2] + 10.107;
   1:  PR[91,3] = PR[90,3] + 3.388;
   1:L PR[91] R[100]mm/sec CNT100;
   1:  PR[91,1] = PR[90,1] + -7.005;
   1:  PR[91,2] = PR[90,2] + 11.087;
   1:  PR[91,3] = PR[90,3] + 3.396;
   1:L PR[91] R[100]mm/sec CNT100;
   1:  PR[91,1] = PR[90,1] + -7.394;
   1:  PR[91,2] = PR[90,2] + 11.549;
   1:  PR[91,3] = PR[90,3] + 3.403;
   1:L PR[91] R[100]mm/sec CNT100;
   1:  PR[91,1] = PR[90,1] + -7.803;
   1:  PR[91,2] = PR[90,2] + 11.999;
   1:  PR[91,3] = PR[90,3] + 3.407;
   1:L PR[91] R[100]mm/sec CNT100;
   1:  PR[91,1] = PR[90,1] + -8.675;
   1:  PR[91,2] = PR[90,2] + 12.863;
   1:  PR[91,3] = PR[90,3] + 3.411;
   1:L PR[91] R[100]mm/sec CNT100;
   1:  PR[91,1] = PR[90,1] + -9.607;
   1:  PR[91,2] = PR[90,2] + 13.660;
   1:  PR[91,3] = PR[90,3] + 3.418;
   1:L PR[91] R[100]mm/sec CNT100;
   1:  PR[91,1] = PR[90,1] + -10.170;
   1:  PR[91,2] = PR[90,2] + 14.087;
   1:  PR[91,3] = PR[90,3] + 3.425;
   1:L PR[91] R[100]mm/sec CNT100;
   1:  PR[91,1] = PR[90,1] + -11.028;
   1:  PR[91,2] = PR[90,2] + 14.672;
   1:  PR[91,3] = PR[90,3] + 3.430;
   1:L PR[91] R[100]mm/sec CNT100;
   1:  PR[91,1] = PR[90,1] + -11.617;
   1:  PR[91,2] = PR[90,2] + 15.033;
   1:  PR[91,3] = PR[90,3] + 3.436;
   1:L PR[91] R[100]mm/sec CNT100;
   1:  PR[91,1] = PR[90,1] + -12.699;
   1:  PR[91,2] = PR[90,2] + 15.611;
   1:  PR[91,3] = PR[90,3] + 3.440;
   1:L PR[91] R[100]mm/sec CNT100;
   1:  PR[91,1] = PR[90,1] + -13.819;
   1:  PR[91,2] = PR[90,2] + 16.109;
   1:  PR[91,3] = PR[90,3] + 3.448;
   1:L PR[91] R[100]mm/sec CNT100;
   1:  PR[91,1] = PR[90,1] + -14.486;
   1:  PR[91,2] = PR[90,2] + 16.359;
   1:  PR[91,3] = PR[90,3] + 3.455;
   1:L PR[91] R[100]mm/sec CNT100;
   1:  PR[91,1] = PR[90,1] + -14.960;
   1:  PR[91,2] = PR[90,2] + 16.521;
   1:  PR[91,3] = PR[90,3] + 3.459;
   1:L PR[91] R[100]mm/sec CNT100;
   1:  PR[91,1] = PR[90,1] + -16.142;
   1:  PR[91,2] = PR[90,2] + 16.852;
   1:  PR[91,3] = PR[90,3] + 3.462;
   1:L PR[91] R[100]mm/sec CNT100;
   1:  PR[91,1] = PR[90,1] + -17.343;
   1:  PR[91,2] = PR[90,2] + 17.098;
   1:  PR[91,3] = PR[90,3] + 3.470;
   1:L PR[91] R[100]mm/sec CNT100;
   1:  PR[91,1] = PR[90,1] + -18.048;
   1:  PR[91,2] = PR[90,2] + 17.198;
   1:  PR[91,3] = PR[90,3] + 3.477;
   1:L PR[91] R[100]mm/sec CNT100;
   1:  PR[91,1] = PR[90,1] + -18.546;
   1:  PR[91,2] = PR[90,2] + 17.254;
   1:  PR[91,3] = PR[90,3] + 3.482;
   1:L PR[91] R[100]mm/sec CNT100;
   1:  PR[91,1] = PR[90,1] + -19.771;
   1:  PR[91,2] = PR[90,2] + 17.324;
   1:  PR[91,3] = PR[90,3] + 3.485;
   1:L PR[91] R[100]mm/sec CNT100;
   1:  PR[91,1] = PR[90,1] + -20.997;
   1:  PR[91,2] = PR[90,2] + 17.304;
   1:  PR[91,3] = PR[90,3] + 3.492;
   1:L PR[91] R[100]mm/sec CNT100;
   1:  PR[91,1] = PR[90,1] + -21.708;
   1:  PR[91,2] = PR[90,2] + 17.251;
   1:  PR[91,3] = PR[90,3] + 3.500;
   1:L PR[91] R[100]mm/sec CNT100;
   1:  PR[91,1] = PR[90,1] + -22.206;
   1:  PR[91,2] = PR[90,2] + 17.198;
   1:  PR[91,3] = PR[90,3] + 3.504;
   1:L PR[91] R[100]mm/sec CNT100;
   1:  PR[91,1] = PR[90,1] + -23.417;
   1:  PR[91,2] = PR[90,2] + 17.002;
   1:  PR[91,3] = PR[90,3] + 3.507;
   1:L PR[91] R[100]mm/sec CNT100;
   1:  PR[91,1] = PR[90,1] + -24.607;
   1:  PR[91,2] = PR[90,2] + 16.720;
   1:  PR[91,3] = PR[90,3] + 3.514;
   1:L PR[91] R[100]mm/sec CNT100;
   1:  PR[91,1] = PR[90,1] + -25.772;
   1:  PR[91,2] = PR[90,2] + 16.354;
   1:  PR[91,3] = PR[90,3] + 3.522;
   1:L PR[91] R[100]mm/sec CNT100;
   1:  PR[91,1] = PR[90,1] + -26.912;
   1:  PR[91,2] = PR[90,2] + 15.902;
   1:  PR[91,3] = PR[90,3] + 3.529;
   1:L PR[91] R[100]mm/sec CNT100;
   1:  PR[91,1] = PR[90,1] + -27.558;
   1:  PR[91,2] = PR[90,2] + 15.601;
   1:  PR[91,3] = PR[90,3] + 3.537;
   1:L PR[91] R[100]mm/sec CNT100;
   1:  PR[91,1] = PR[90,1] + -28.008;
   1:  PR[91,2] = PR[90,2] + 15.373;
   1:  PR[91,3] = PR[90,3] + 3.541;
   1:L PR[91] R[100]mm/sec CNT100;
   1:  PR[91,1] = PR[90,1] + -28.635;
   1:  PR[91,2] = PR[90,2] + 15.023;
   1:  PR[91,3] = PR[90,3] + 3.544;
   1:L PR[91] R[100]mm/sec CNT100;
   1:  PR[91,1] = PR[90,1] + -29.069;
   1:  PR[91,2] = PR[90,2] + 14.763;
   1:  PR[91,3] = PR[90,3] + 3.549;
   1:L PR[91] R[100]mm/sec CNT100;
   1:  PR[91,1] = PR[90,1] + -29.579;
   1:  PR[91,2] = PR[90,2] + 14.432;
   1:  PR[91,3] = PR[90,3] + 3.552;
   1:L PR[91] R[100]mm/sec CNT100;
   1:  PR[91,1] = PR[90,1] + -30.077;
   1:  PR[91,2] = PR[90,2] + 14.082;
   1:  PR[91,3] = PR[90,3] + 3.555;
   1:L PR[91] R[100]mm/sec CNT100;
   1:  PR[91,1] = PR[90,1] + -31.042;
   1:  PR[91,2] = PR[90,2] + 13.323;
   1:  PR[91,3] = PR[90,3] + 3.559;
   1:L PR[91] R[100]mm/sec CNT100;
   1:  PR[91,1] = PR[90,1] + -31.948;
   1:  PR[91,2] = PR[90,2] + 12.497;
   1:  PR[91,3] = PR[90,3] + 3.566;
   1:L PR[91] R[100]mm/sec CNT100;
   1:  PR[91,1] = PR[90,1] + -32.441;
   1:  PR[91,2] = PR[90,2] + 11.991;
   1:  PR[91,3] = PR[90,3] + 3.574;
   1:L PR[91] R[100]mm/sec CNT100;
   1:  PR[91,1] = PR[90,1] + -33.131;
   1:  PR[91,2] = PR[90,2] + 11.210;
   1:  PR[91,3] = PR[90,3] + 3.578;
   1:L PR[91] R[100]mm/sec CNT100;
   1:  PR[91,1] = PR[90,1] + -33.560;
   1:  PR[91,2] = PR[90,2] + 10.672;
   1:  PR[91,3] = PR[90,3] + 3.585;
   1:L PR[91] R[100]mm/sec CNT100;
   1:  PR[91,1] = PR[90,1] + -34.267;
   1:  PR[91,2] = PR[90,2] + 9.671;
   1:  PR[91,3] = PR[90,3] + 3.589;
   1:L PR[91] R[100]mm/sec CNT100;
   1:  PR[91,1] = PR[90,1] + -34.898;
   1:  PR[91,2] = PR[90,2] + 8.625;
   1:  PR[91,3] = PR[90,3] + 3.596;
   1:L PR[91] R[100]mm/sec CNT100;
   1:  PR[91,1] = PR[90,1] + -35.454;
   1:  PR[91,2] = PR[90,2] + 7.531;
   1:  PR[91,3] = PR[90,3] + 3.604;
   1:L PR[91] R[100]mm/sec CNT100;
   1:  PR[91,1] = PR[90,1] + -35.738;
   1:  PR[91,2] = PR[90,2] + 6.877;
   1:  PR[91,3] = PR[90,3] + 3.611;
   1:L PR[91] R[100]mm/sec CNT100;
   1:  PR[91,1] = PR[90,1] + -35.926;
   1:  PR[91,2] = PR[90,2] + 6.408;
   1:  PR[91,3] = PR[90,3] + 3.615;
   1:L PR[91] R[100]mm/sec CNT100;
   1:  PR[91,1] = PR[90,1] + -36.137;
   1:  PR[91,2] = PR[90,2] + 5.815;
   1:  PR[91,3] = PR[90,3] + 3.618;
   1:L PR[91] R[100]mm/sec CNT100;
   1:  PR[91,1] = PR[90,1] + -36.315;
   1:  PR[91,2] = PR[90,2] + 5.255;
   1:  PR[91,3] = PR[90,3] + 3.622;
   1:L PR[91] R[100]mm/sec CNT100;
   1:  PR[91,1] = PR[90,1] + -36.622;
   1:  PR[91,2] = PR[90,2] + 4.066;
   1:  PR[91,3] = PR[90,3] + 3.626;
   1:L PR[91] R[100]mm/sec CNT100;
   1:  PR[91,1] = PR[90,1] + -36.843;
   1:  PR[91,2] = PR[90,2] + 2.858;
   1:  PR[91,3] = PR[90,3] + 3.633;
   1:L PR[91] R[100]mm/sec CNT100;
   1:  PR[91,1] = PR[90,1] + -36.975;
   1:  PR[91,2] = PR[90,2] + 1.650;
   1:  PR[91,3] = PR[90,3] + 3.641;
   1:L PR[91] R[100]mm/sec CNT100;
   1:  PR[91,1] = PR[90,1] + -37.019;
   1:  PR[91,2] = PR[90,2] + 0.422;
   1:  PR[91,3] = PR[90,3] + 3.648;
   1:L PR[91] R[100]mm/sec CNT100;
   1:  PR[91,1] = PR[90,1] + -37.009;
   1:  PR[91,2] = PR[90,2] + -0.164;
   1:  PR[91,3] = PR[90,3] + 3.656;
   1:L PR[91] R[100]mm/sec CNT100;
   1:  PR[91,1] = PR[90,1] + -36.975;
   1:  PR[91,2] = PR[90,2] + -0.793;
   1:  PR[91,3] = PR[90,3] + 3.659;
   1:L PR[91] R[100]mm/sec CNT100;
   1:  PR[91,1] = PR[90,1] + -36.906;
   1:  PR[91,2] = PR[90,2] + -1.507;
   1:  PR[91,3] = PR[90,3] + 3.663;
   1:L PR[91] R[100]mm/sec CNT100;
   1:  PR[91,1] = PR[90,1] + -36.843;
